C07281=1141.600,42.960,-51.075,-179.900,6.400,149.135
C07282=1141.605,42.711,-51.060,-179.904,6.398,149.135
C07283=1141.610,42.462,-51.044,-179.906,6.397,149.136
C07284=1141.615,42.212,-51.029,-179.909,6.396,149.136
C07285=1141.621,41.962,-51.014,-179.911,6.395,149.137
C07286=1141.625,41.713,-50.999,-179.914,6.394,149.138
C07287=1141.630,41.463,-50.983,-179.916,6.393,149.138
C07288=1141.635,41.214,-50.969,-179.919,6.392,149.139
C07289=1141.641,40.964,-50.953,-179.922,6.391,149.139
C07290=1141.645,40.715,-50.938,-179.924,6.390,149.140
C07291=1141.651,40.466,-50.923,-179.927,6.389,149.140
C07292=1141.656,40.216,-50.908,-179.929,6.388,149.141
C07293=1141.660,39.967,-50.893,-179.932,6.387,149.141
C07294=1141.666,39.717,-50.878,-179.935,6.386,149.142
C07295=1141.671,39.468,-50.864,-179.937,6.384,149.142
C07296=1141.676,39.218,-50.848,-179.940,6.384,149.143
C07297=1141.680,38.969,-50.833,-179.943,6.382,149.143
C07298=1141.686,38.718,-50.818,-179.945,6.381,149.144
C07299=1141.690,38.469,-50.803,-179.948,6.380,149.144
C07300=1141.696,38.219,-50.788,-179.950,6.379,149.145
C07301=1141.701,37.970,-50.773,-179.953,6.379,149.146
C07302=1141.705,37.721,-50.758,-179.956,6.377,149.146
C07303=1141.711,37.471,-50.743,-179.958,6.376,149.146
C07304=1141.716,37.222,-50.728,-179.961,6.375,149.147
C07305=1141.721,36.972,-50.713,-179.963,6.374,149.148
C07306=1141.726,36.723,-50.698,-179.966,6.372,149.148
C07307=1141.731,36.473,-50.684,-179.969,6.372,149.149
C07308=1141.736,36.224,-50.668,-179.971,6.370,149.149
C07309=1141.741,35.974,-50.654,-179.974,6.370,149.150
C07310=1141.746,35.725,-50.639,-179.976,6.369,149.150
C07311=1141.752,35.475,-50.624,-179.979,6.367,149.151
C07312=1141.756,35.226,-50.609,-179.982,6.367,149.151
C07313=1141.761,34.976,-50.595,-179.984,6.365,149.152
C07314=1141.767,34.727,-50.579,-179.987,6.365,149.152
C07315=1141.772,34.477,-50.565,-179.989,6.364,149.153
C07316=1141.776,34.228,-50.550,-179.992,6.362,149.153
C07317=1141.782,33.978,-50.535,-179.994,6.362,149.154
C07318=1141.787,33.729,-50.520,-179.997,6.360,149.155
C07319=1141.792,33.479,-50.506,-180.000,6.360,149.155
C07320=1141.797,33.230,-50.490,179.997,6.358,149.156
C07321=1141.802,32.980,-50.476,179.995,6.357,149.156
C07322=1141.807,32.730,-50.462,179.993,6.357,149.157
C07323=1141.812,32.481,-50.447,179.990,6.355,149.157
C07324=1141.817,32.231,-50.432,179.987,6.355,149.158
C07325=1141.822,31.983,-50.417,179.985,6.353,149.158
C07326=1141.827,31.733,-50.403,179.982,6.352,149.159
C07327=1141.832,31.483,-50.389,179.980,6.352,149.159
C07328=1141.838,31.234,-50.373,179.977,6.350,149.160
C07329=1141.843,30.984,-50.359,179.974,6.350,149.160
C07330=1141.848,30.735,-50.345,179.972,6.348,149.161
C07331=1141.852,30.486,-50.330,179.969,6.348,149.162
C07332=1141.858,30.236,-50.315,179.967,6.347,149.162
C07333=1141.863,29.986,-50.300,179.964,6.345,149.162
C07334=1141.868,29.737,-50.285,179.961,6.345,149.163
C07335=1141.873,29.487,-50.271,179.959,6.343,149.164
C07336=1141.878,29.237,-50.257,179.956,6.343,149.164
C07337=1141.884,28.988,-50.242,179.954,6.342,149.165
C07338=1141.888,28.739,-50.227,179.951,6.340,149.165
C07339=1141.893,28.489,-50.213,179.948,6.340,149.166
C07340=1141.898,28.239,-50.199,179.946,6.339,149.166
C07341=1141.903,27.990,-50.185,179.943,6.338,149.167
C07342=1141.908,27.721,-50.169,179.941,6.337,149.167
C07343=1141.914,27.452,-50.152,179.938,6.335,149.168
C07344=1141.920,27.182,-50.138,179.935,6.334,149.169
C07345=1141.925,26.914,-50.122,179.932,6.333,149.169
C07346=1141.930,26.665,-50.108,179.930,6.333,149.170
C07347=1141.935,26.415,-50.094,179.927,6.331,149.170
C07348=1141.940,26.166,-50.079,179.925,6.331,149.171
C07349=1141.946,25.916,-50.064,179.922,6.329,149.171
C07350=1141.951,25.666,-50.049,179.919,6.328,149.172
C07351=1141.956,25.416,-50.035,179.917,6.328,149.172
C07352=1141.961,25.167,-50.021,179.914,6.326,149.173
C07353=1141.966,24.918,-50.007,179.912,6.326,149.174
C07354=1141.971,24.668,-49.993,179.910,6.325,149.174
C07355=1141.976,24.418,-49.978,179.906,6.323,149.175
C07356=1141.981,24.169,-49.964,179.904,6.323,149.175
C07357=1141.986,23.920,-49.950,179.902,6.322,149.176
C07358=1141.991,23.670,-49.935,179.899,6.321,149.176
C07359=1141.996,23.421,-49.921,179.897,6.320,149.177
C07360=1142.001,23.171,-49.907,179.894,6.319,149.177
C07361=1142.006,22.921,-49.892,179.891,6.318,149.178
C07362=1142.012,22.672,-49.879,179.889,6.317,149.178
C07363=1142.017,22.423,-49.864,179.886,6.316,149.179
C07364=1142.022,22.173,-49.850,179.884,6.315,149.180
C07365=1142.027,21.923,-49.836,179.881,6.314,149.180
C07366=1142.032,21.674,-49.822,179.879,6.314,149.181
C07367=1142.037,21.424,-49.808,179.876,6.312,149.181
C07368=1142.042,21.175,-49.793,179.873,6.311,149.182
C07369=1142.047,20.925,-49.779,179.871,6.311,149.182
C07370=1142.052,20.675,-49.765,179.868,6.309,149.183
C07371=1142.057,20.426,-49.751,179.866,6.309,149.183
C07372=1142.062,20.177,-49.736,179.864,6.308,149.184
C07373=1142.067,19.927,-49.722,179.860,6.307,149.185
C07374=1142.073,19.677,-49.709,179.858,6.306,149.185
C07375=1142.078,19.428,-49.695,179.856,6.305,149.185
C07376=1142.083,19.178,-49.680,179.853,6.304,149.186
C07377=1142.088,18.928,-49.666,179.851,6.303,149.187
C07378=1142.094,18.679,-49.652,179.848,6.302,149.187
C07379=1142.099,18.429,-49.638,179.845,6.301,149.188
C07380=1142.103,18.180,-49.624,179.843,6.300,149.188
C07381=1142.108,17.931,-49.610,179.840,6.299,149.189
C07382=1142.113,17.681,-49.596,179.837,6.298,149.189
C07383=1142.119,17.431,-49.583,179.835,6.297,149.190
C07384=1142.124,17.181,-49.568,179.833,6.297,149.190
C07385=1142.129,16.932,-49.554,179.831,6.296,149.191
C07386=1142.134,16.683,-49.540,179.827,6.295,149.192
C07387=1142.139,16.433,-49.526,179.825,6.294,149.192
C07388=1142.144,16.184,-49.513,179.822,6.293,149.193
C07389=1142.149,15.934,-49.499,179.820,6.292,149.193
C07390=1142.154,15.684,-49.485,179.817,6.291,149.194
C07391=1142.160,15.435,-49.471,179.815,6.290,149.194
C07392=1142.165,15.185,-49.456,179.813,6.290,149.195
C07393=1142.170,14.935,-49.443,179.809,6.288,149.195
C07394=1142.175,14.686,-49.430,179.807,6.288,149.196
C07395=1142.180,14.437,-49.415,179.805,6.287,149.196
C07396=1142.185,14.188,-49.401,179.802,6.286,149.197
C07397=1142.190,13.937,-49.388,179.800,6.285,149.198
C07398=1142.195,13.688,-49.374,179.797,6.284,149.198
C07399=1142.200,13.439,-49.360,179.795,6.283,149.199
C07400=1142.205,13.189,-49.347,179.792,6.282,149.199
C07401=1142.210,12.939,-49.332,179.789,6.281,149.200
C07402=1142.216,12.690,-49.319,179.787,6.281,149.200
C07403=1142.220,12.440,-49.306,179.784,6.279,149.201
C07404=1142.226,12.191,-49.292,179.782,6.279,149.201
C07405=1142.231,11.941,-49.277,179.780,6.278,149.202
C07406=1142.236,11.691,-49.264,179.777,6.277,149.203
C07407=1142.241,11.442,-49.250,179.774,6.276,149.203
C07408=1142.246,11.192,-49.236,179.772,6.275,149.204
C07409=1142.252,10.943,-49.223,179.769,6.274,149.204
C07410=1142.256,10.693,-49.209,179.767,6.274,149.205
C07411=1142.261,10.443,-49.196,179.764,6.272,149.205
C07412=1142.267,10.194,-49.182,179.762,6.272,149.206
C07413=1142.272,9.944,-49.168,179.759,6.271,149.206
C07414=1142.277,9.695,-49.155,179.757,6.270,149.207
C07415=1142.282,9.445,-49.141,179.754,6.269,149.207
C07416=1142.288,9.196,-49.127,179.752,6.268,149.208
C07417=1142.292,8.946,-49.114,179.749,6.267,149.209
C07418=1142.298,8.697,-49.101,179.747,6.267,149.209
C07419=1142.303,8.447,-49.086,179.744,6.265,149.210
C07420=1142.307,8.197,-49.073,179.742,6.265,149.210
C07421=1142.313,7.948,-49.059,179.739,6.264,149.211
C07422=1142.318,7.698,-49.046,179.737,6.263,149.211
C07423=1142.323,7.449,-49.033,179.734,6.262,149.212
C07424=1142.328,7.198,-49.019,179.732,6.261,149.212
C07425=1142.333,6.950,-49.006,179.729,6.260,149.213
C07426=1142.338,6.699,-48.992,179.727,6.260,149.214
C07427=1142.344,6.450,-48.978,179.724,6.258,149.214
C07428=1142.348,6.200,-48.965,179.721,6.258,149.215
C07429=1142.354,5.951,-48.951,179.719,6.257,149.215
C07430=1142.358,5.701,-48.938,179.717,6.256,149.216
C07431=1142.364,5.452,-48.925,179.714,6.255,149.216
C07432=1142.369,5.202,-48.911,179.711,6.254,149.217
C07433=1142.374,4.953,-48.898,179.709,6.254,149.218
C07434=1142.379,4.703,-48.884,179.707,6.253,149.218
C07435=1142.384,4.454,-48.871,179.704,6.252,149.218
C07436=1142.390,4.203,-48.858,179.701,6.251,149.219
C07437=1142.395,3.955,-48.845,179.699,6.250,149.220
C07438=1142.400,3.704,-48.831,179.696,6.250,149.220
C07439=1142.405,3.455,-48.818,179.694,6.249,149.221
C07440=1142.410,3.205,-48.804,179.692,6.249,149.221
C07441=1142.415,2.956,-48.792,179.689,6.247,149.222
C07442=1142.421,2.706,-48.778,179.687,6.246,149.222
C07443=1142.425,2.457,-48.765,179.684,6.246,149.223
C07444=1142.431,2.207,-48.751,179.682,6.245,149.224
C07445=1142.435,1.957,-48.738,179.679,6.244,149.224
C07446=1142.442,1.689,-48.724,179.676,6.243,149.225
C07447=1142.447,1.419,-48.710,179.674,6.242,149.225
C07448=1142.453,1.149,-48.695,179.671,6.241,149.226
C07449=1142.458,0.879,-48.681,179.668,6.240,149.227
C07450=1142.464,0.630,-48.668,179.666,6.240,149.227
C07451=1142.468,0.381,-48.654,179.663,6.239,149.228
C07452=1142.474,0.131,-48.641,179.661,6.238,149.228
C07453=1142.479,-0.119,-48.628,179.658,6.237,149.229
C07454=1142.483,-0.369,-48.615,179.656,6.236,149.229
C07455=1142.489,-0.618,-48.602,179.654,6.235,149.230
C07456=1142.494,-0.867,-48.589,179.651,6.235,149.230
C07457=1142.499,-1.117,-48.575,179.648,6.233,149.231
C07458=1142.504,-1.367,-48.563,179.646,6.233,149.232
C07459=1142.510,-1.617,-48.549,179.643,6.232,149.232
C07460=1142.515,-1.866,-48.536,179.641,6.231,149.233
C07461=1142.520,-2.115,-48.523,179.639,6.231,149.233
C07462=1142.525,-2.365,-48.510,179.636,6.230,149.234
C07463=1142.530,-2.615,-48.497,179.633,6.229,149.234
C07464=1142.536,-2.864,-48.484,179.631,6.228,149.235
C07465=1142.540,-3.114,-48.471,179.629,6.227,149.235
C07466=1142.545,-3.363,-48.458,179.626,6.227,149.236
C07467=1142.551,-3.613,-48.445,179.624,6.226,149.236
C07468=1142.556,-3.863,-48.432,179.621,6.226,149.237
C07469=1142.561,-4.112,-48.419,179.619,6.224,149.238
C07470=1142.567,-4.361,-48.406,179.616,6.223,149.238
C07471=1142.571,-4.611,-48.393,179.614,6.223,149.239
C07472=1142.576,-4.861,-48.380,179.611,6.222,149.239
C07473=1142.582,-5.110,-48.367,179.609,6.222,149.240
C07474=1142.587,-5.360,-48.354,179.607,6.221,149.240
C07475=1142.592,-5.610,-48.341,179.604,6.219,149.241
C07476=1142.598,-5.859,-48.328,179.601,6.219,149.242
C07477=1142.602,-6.109,-48.315,179.599,6.218,149.242
C07478=1142.607,-6.359,-48.302,179.596,6.218,149.243
C07479=1142.613,-6.608,-48.289,179.594,6.217,149.243
C07480=1142.618,-6.858,-48.276,179.592,6.216,149.244
C07481=1142.623,-7.108,-48.264,179.589,6.216,149.244
C07482=1142.628,-7.357,-48.251,179.587,6.214,149.245
C07483=1142.634,-7.607,-48.238,179.584,6.214,149.245
C07484=1142.638,-7.857,-48.225,179.582,6.213,149.246
C07485=1142.643,-8.106,-48.212,179.580,6.212,149.246
C07486=1142.648,-8.355,-48.200,179.577,6.211,149.247
C07487=1142.654,-8.605,-48.186,179.575,6.211,149.248
C07488=1142.659,-8.855,-48.174,179.572,6.210,149.248
C07489=1142.664,-9.105,-48.162,179.569,6.209,149.249
C07490=1142.669,-9.354,-48.149,179.567,6.208,149.249
C07491=1142.675,-9.605,-48.135,179.564,6.207,149.250
C07492=1142.680,-9.854,-48.123,179.562,6.207,149.250
C07493=1142.685,-10.103,-48.110,179.560,6.206,149.251
C07494=1142.690,-10.352,-48.098,179.557,6.205,149.252
C07495=1142.695,-10.602,-48.085,179.555,6.205,149.252
C07496=1142.700,-10.852,-48.072,179.553,6.204,149.253
C07497=1142.706,-11.101,-48.059,179.550,6.203,149.253
C07498=1142.711,-11.351,-48.047,179.547,6.202,149.254
C07499=1142.716,-11.601,-48.034,179.545,6.201,149.254
C07500=1142.721,-11.851,-48.021,179.542,6.201,149.255
C07501=1142.726,-12.100,-48.009,179.540,6.200,149.255
C07502=1142.731,-12.349,-47.996,179.538,6.199,149.256
C07503=1142.737,-12.600,-47.984,179.535,6.199,149.257
C07504=1142.742,-12.849,-47.971,179.533,6.198,149.257
C07505=1142.747,-13.099,-47.958,179.530,6.198,149.258
C07506=1142.752,-13.348,-47.946,179.528,6.196,149.258
C07507=1142.757,-13.598,-47.933,179.526,6.195,149.259
C07508=1142.762,-13.847,-47.921,179.523,6.195,149.259
C07509=1142.767,-14.097,-47.909,179.521,6.194,149.260
C07510=1142.772,-14.347,-47.896,179.518,6.194,149.261
C07511=1142.778,-14.596,-47.882,179.516,6.193,149.261
C07512=1142.783,-14.846,-47.870,179.514,6.192,149.262
C07513=1142.788,-15.096,-47.858,179.511,6.192,149.262
C07514=1142.794,-15.345,-47.845,179.509,6.191,149.263
C07515=1142.799,-15.595,-47.833,179.506,6.190,149.263
C07516=1142.803,-15.845,-47.820,179.504,6.190,149.264
C07517=1142.809,-16.094,-47.808,179.501,6.188,149.264
C07518=1142.814,-16.344,-47.796,179.499,6.188,149.265
C07519=1142.819,-16.594,-47.783,179.496,6.187,149.265
C07520=1142.824,-16.843,-47.771,179.494,6.186,149.266
C07521=1142.830,-17.093,-47.759,179.492,6.186,149.267
C07522=1142.835,-17.342,-47.746,179.489,6.185,149.267
C07523=1142.840,-17.591,-47.734,179.487,6.184,149.268
C07524=1142.845,-17.842,-47.721,179.485,6.184,149.268
C07525=1142.850,-18.091,-47.709,179.482,6.183,149.269
C07526=1142.855,-18.341,-47.696,179.480,6.182,149.269
C07527=1142.860,-18.591,-47.684,179.477,6.182,149.270
C07528=1142.866,-18.840,-47.672,179.475,6.181,149.271
C07529=1142.871,-19.090,-47.660,179.472,6.180,149.271
C07530=1142.876,-19.339,-47.647,179.469,6.179,149.272
C07531=1142.881,-19.589,-47.635,179.467,6.178,149.272
C07532=1142.887,-19.838,-47.623,179.465,6.178,149.273
C07533=1142.892,-20.088,-47.610,179.462,6.177,149.273
C07534=1142.897,-20.338,-47.598,179.460,6.176,149.274
C07535=1142.902,-20.588,-47.585,179.458,6.176,149.275
C07536=1142.907,-20.838,-47.573,179.455,6.175,149.275
C07537=1142.912,-21.087,-47.561,179.453,6.174,149.276
C07538=1142.918,-21.337,-47.549,179.450,6.174,149.276
C07539=1142.923,-21.586,-47.536,179.448,6.173,149.277
C07540=1142.928,-21.836,-47.524,179.446,6.173,149.277
C07541=1142.933,-22.086,-47.512,179.443,6.172,149.278
C07542=1142.939,-22.335,-47.500,179.441,6.171,149.278
C07543=1142.944,-22.585,-47.487,179.439,6.171,149.279
C07544=1142.949,-22.835,-47.475,179.436,6.170,149.280
C07545=1142.955,-23.084,-47.463,179.434,6.170,149.280
C07546=1142.959,-23.334,-47.452,179.432,6.169,149.281
C07547=1142.965,-23.584,-47.440,179.429,6.167,149.281
C07548=1142.970,-23.833,-47.427,179.426,6.167,149.282
C07549=1142.975,-24.083,-47.415,179.424,6.166,149.282
C07550=1142.980,-24.353,-47.402,179.421,6.166,149.283
C07551=1142.987,-24.623,-47.388,179.419,6.165,149.283
C07552=1142.992,-24.893,-47.375,179.416,6.164,149.284
C07553=1142.997,-25.163,-47.362,179.414,6.164,149.285
C07554=1143.003,-25.413,-47.350,179.412,6.163,149.285
C07555=1143.008,-25.662,-47.338,179.409,6.162,149.286
C07556=1143.013,-25.912,-47.327,179.407,6.162,149.287
C07557=1143.018,-26.161,-47.314,179.404,6.160,149.287
C07558=1143.023,-26.411,-47.302,179.402,6.160,149.287
C07559=1143.029,-26.661,-47.290,179.399,6.159,149.288
C07560=1143.034,-26.911,-47.278,179.397,6.158,149.289
C07561=1143.039,-27.160,-47.266,179.394,6.158,149.289
C07562=1143.044,-27.410,-47.254,179.392,6.157,149.290
C07563=1143.049,-27.659,-47.242,179.390,6.156,149.290
C07564=1143.054,-27.909,-47.230,179.387,6.156,149.291
C07565=1143.061,-28.159,-47.218,179.385,6.155,149.291
C07566=1143.065,-28.408,-47.207,179.382,6.155,149.292
C07567=1143.070,-28.658,-47.195,179.380,6.154,149.293
C07568=1143.076,-28.908,-47.183,179.378,6.153,149.293
C07569=1143.081,-29.157,-47.171,179.375,6.153,149.294
C07570=1143.086,-29.407,-47.160,179.373,6.152,149.294
C07571=1143.091,-29.656,-47.147,179.371,6.151,149.295
C07572=1143.096,-29.906,-47.135,179.368,6.151,149.295
C07573=1143.102,-30.156,-47.123,179.366,6.150,149.296
C07574=1143.107,-30.406,-47.112,179.363,6.150,149.297
C07575=1143.112,-30.655,-47.099,179.361,6.149,149.297
C07576=1143.117,-30.905,-47.087,179.359,6.148,149.298
C07577=1143.123,-31.155,-47.075,179.356,6.148,149.298
C07578=1143.127,-31.405,-47.064,179.354,6.147,149.299
C07579=1143.133,-31.655,-47.052,179.352,6.146,149.299
C07580=1143.138,-31.903,-47.040,179.349,6.146,149.300
C07581=1143.143,-32.153,-47.029,179.347,6.145,149.300
C07582=1143.149,-32.403,-47.017,179.345,6.144,149.301
C07583=1143.154,-32.653,-47.005,179.342,6.144,149.302
C07584=1143.159,-32.902,-46.994,179.340,6.143,149.302
C07585=1143.164,-33.152,-46.982,179.338,6.142,149.303
C07586=1143.170,-33.402,-46.970,179.335,6.142,149.303
C07587=1143.174,-33.651,-46.958,179.333,6.141,149.304
C07588=1143.180,-33.901,-46.946,179.331,6.140,149.304
C07589=1143.185,-34.150,-46.935,179.328,6.140,149.305
C07590=1143.190,-34.400,-46.923,179.326,6.139,149.306
C07591=1143.195,-34.650,-46.911,179.323,6.138,149.306
C07592=1143.201,-34.900,-46.899,179.322,6.138,149.306
C07593=1143.206,-35.150,-46.888,179.319,6.138,149.307
C07594=1143.211,-35.400,-46.876,179.317,6.137,149.308
C07595=1143.217,-35.649,-46.865,179.314,6.137,149.308
C07596=1143.222,-35.898,-46.853,179.312,6.136,149.309
C07597=1143.227,-36.148,-46.842,179.310,6.135,149.309
C07598=1143.232,-36.398,-46.830,179.307,6.135,149.310
C07599=1143.237,-36.648,-46.818,179.305,6.134,149.310
C07600=1143.243,-36.898,-46.807,179.302,6.134,149.311
C07601=1143.248,-37.147,-46.796,179.300,6.133,149.312
C07602=1143.253,-37.397,-46.784,179.298,6.132,149.312
C07603=1143.258,-37.646,-46.772,179.295,6.132,149.313
C07604=1143.264,-37.896,-46.761,179.293,6.131,149.313
C07605=1143.268,-38.146,-46.749,179.291,6.130,149.314
C07606=1143.274,-38.395,-46.738,179.288,6.130,149.314
C07607=1143.280,-38.645,-46.726,179.286,6.129,149.315
C07608=1143.284,-38.895,-46.715,179.284,6.128,149.315
C07609=1143.290,-39.145,-46.703,179.281,6.128,149.316
C07610=1143.295,-39.394,-46.691,179.279,6.127,149.317
C07611=1143.301,-39.643,-46.680,179.277,6.127,149.317
C07612=1143.305,-39.893,-46.669,179.274,6.126,149.318
C07613=1143.311,-40.143,-46.657,179.272,6.125,149.318
C07614=1143.315,-40.393,-46.645,179.269,6.125,149.319
C07615=1143.321,-40.642,-46.634,179.268,6.125,149.319
C07616=1143.326,-40.892,-46.623,179.266,6.124,149.320
C07617=1143.332,-41.142,-46.611,179.263,6.123,149.321
C07618=1143.337,-41.392,-46.600,179.261,6.123,149.321
C07619=1143.343,-41.641,-46.589,179.258,6.122,149.322
C07620=1143.347,-41.891,-46.577,179.256,6.121,149.322
C07621=1143.353,-42.141,-46.565,179.254,6.121,149.323
C07622=1143.357,-42.390,-46.554,179.251,6.120,149.323
C07623=1143.364,-42.640,-46.543,179.249,6.120,149.324
C07624=1143.368,-42.890,-46.532,179.247,6.119,149.324
C07625=1143.374,-43.140,-46.520,179.244,6.118,149.325
C07626=1143.379,-43.389,-46.509,179.242,6.118,149.326
C07627=1143.384,-43.638,-46.498,179.240,6.117,149.326
C07628=1143.389,-43.888,-46.486,179.237,6.116,149.327
C07629=1143.394,-44.138,-46.476,179.235,6.116,149.327
C07630=1143.400,-44.388,-46.464,179.233,6.116,149.328
C07631=1143.405,-44.637,-46.453,179.231,6.115,149.328
C07632=1143.410,-44.887,-46.441,179.228,6.114,149.329
C07633=1143.415,-45.137,-46.430,179.226,6.114,149.330
C07634=1143.421,-45.386,-46.419,179.224,6.113,149.330
C07635=1143.426,-45.636,-46.407,179.221,6.112,149.331
C07636=1143.431,-45.886,-46.396,179.219,6.112,149.331
C07637=1143.436,-46.135,-46.386,179.217,6.111,149.332
C07638=1143.442,-46.385,-46.374,179.214,6.111,149.332
C07639=1143.447,-46.635,-46.363,179.212,6.110,149.333
C07640=1143.453,-46.884,-46.351,179.210,6.109,149.333
C07641=1143.458,-47.134,-46.341,179.207,6.110,149.334
C07642=1143.462,-47.384,-46.329,179.205,6.109,149.335
C07643=1143.468,-47.633,-46.318,179.203,6.108,149.335
C07644=1143.473,-47.883,-46.307,179.200,6.108,149.336
C07645=1143.478,-48.133,-46.296,179.198,6.107,149.336
C07646=1143.484,-48.382,-46.284,179.196,6.106,149.337
C07647=1143.489,-48.633,-46.274,179.193,6.106,149.337
C07648=1143.494,-48.882,-46.263,179.191,6.105,149.338
C07649=1143.500,-49.132,-46.252,179.189,6.104,149.338
C07650=1143.505,-49.382,-46.241,179.186,6.104,149.339
C07651=1143.509,-49.631,-46.229,179.185,6.104,149.340
C07652=1143.516,-49.881,-46.218,179.183,6.103,149.340
C07653=1143.520,-50.131,-46.207,179.180,6.103,149.341
C07654=1143.527,-50.401,-46.195,179.178,6.102,149.341
C07655=1143.532,-50.672,-46.184,179.175,6.102,149.342
C07656=1143.537,-50.943,-46.171,179.173,6.101,149.342
C07657=1143.543,-51.213,-46.159,179.170,6.100,149.343
C07658=1143.548,-51.463,-46.149,179.168,6.100,149.344
C07659=1143.554,-51.713,-46.137,179.165,6.099,149.344
C07660=1143.559,-51.963,-46.127,179.163,6.098,149.345
C07661=1143.564,-52.212,-46.115,179.161,6.098,149.345
C07662=1143.570,-52.462,-46.105,179.158,6.097,149.346
C07663=1143.575,-52.712,-46.093,179.156,6.096,149.346
C07664=1143.580,-52.961,-46.082,179.154,6.096,149.347
C07665=1143.585,-53.211,-46.072,179.152,6.096,149.348
C07666=1143.590,-53.461,-46.061,179.150,6.095,149.348
C07667=1143.596,-53.710,-46.050,179.147,6.095,149.349
C07668=1143.601,-53.960,-46.039,179.145,6.094,149.349
C07669=1143.607,-54.210,-46.028,179.143,6.093,149.350
C07670=1143.612,-54.460,-46.018,179.140,6.093,149.350
C07671=1143.616,-54.710,-46.006,179.138,6.092,149.351
C07672=1143.622,-54.959,-45.996,179.136,6.092,149.351
C07673=1143.627,-55.209,-45.984,179.134,6.091,149.352
C07674=1143.633,-55.459,-45.974,179.131,6.091,149.353
C07675=1143.638,-55.708,-45.963,179.129,6.090,149.353
C07676=1143.643,-55.958,-45.953,179.127,6.090,149.354
C07677=1143.648,-56.207,-45.941,179.124,6.089,149.354
C07678=1143.654,-56.457,-45.931,179.123,6.089,149.355
C07679=1143.659,-56.707,-45.920,179.120,6.088,149.355
C07680=1143.664,-56.957,-45.909,179.118,6.088,149.356
C07681=1143.670,-57.207,-45.898,179.116,6.087,149.356
C07682=1143.674,-57.456,-45.887,179.113,6.086,149.357
C07683=1143.680,-57.706,-45.877,179.111,6.086,149.358
C07684=1143.685,-57.956,-45.866,179.109,6.085,149.358
C07685=1143.690,-58.205,-45.855,179.107,6.085,149.359
C07686=1143.695,-58.455,-45.845,179.104,6.085,149.359
C07687=1143.701,-58.705,-45.835,179.102,6.084,149.360
C07688=1143.706,-58.955,-45.823,179.100,6.083,149.360
C07689=1143.712,-59.204,-45.813,179.097,6.083,149.361
C07690=1143.717,-59.454,-45.801,179.095,6.082,149.361
C07691=1143.722,-59.703,-45.791,179.093,6.082,149.362
C07692=1143.727,-59.954,-45.781,179.091,6.082,149.363
C07693=1143.733,-60.203,-45.770,179.089,6.081,149.363
C07694=1143.737,-60.453,-45.759,179.086,6.080,149.364
C07695=1143.743,-60.702,-45.749,179.084,6.080,149.364
C07696=1143.748,-60.953,-45.738,179.082,6.079,149.365
C07697=1143.753,-61.202,-45.727,179.080,6.079,149.365
C07698=1143.758,-61.452,-45.717,179.077,6.079,149.366
C07699=1143.764,-61.701,-45.707,179.075,6.078,149.366
C07700=1143.769,-61.951,-45.696,179.073,6.077,149.367
C07701=1143.774,-62.200,-45.685,179.070,6.077,149.368
C07702=1143.780,-62.450,-45.675,179.069,6.077,149.368
C07703=1143.785,-62.700,-45.664,179.066,6.076,149.369
C07704=1143.790,-62.950,-45.654,179.064,6.076,149.369
C07705=1143.795,-63.199,-45.643,179.062,6.075,149.370
C07706=1143.801,-63.449,-45.633,179.059,6.074,149.370
C07707=1143.806,-63.699,-45.622,179.057,6.073,149.371
C07708=1143.811,-63.949,-45.612,179.055,6.074,149.371
C07709=1143.817,-64.198,-45.602,179.053,6.073,149.372
C07710=1143.822,-64.448,-45.590,179.051,6.072,149.372
C07711=1143.827,-64.697,-45.580,179.048,6.072,149.373
C07712=1143.832,-64.948,-45.569,179.046,6.071,149.374
C07713=1143.838,-65.197,-45.559,179.044,6.071,149.374
C07714=1143.843,-65.448,-45.549,179.042,6.071,149.375
C07715=1143.848,-65.697,-45.538,179.039,6.070,149.375
C07716=1143.854,-65.947,-45.528,179.037,6.069,149.376
C07717=1143.859,-66.196,-45.517,179.035,6.069,149.376
C07718=1143.864,-66.446,-45.507,179.033,6.069,149.377
C07719=1143.869,-66.696,-45.496,179.031,6.068,149.377
C07720=1143.875,-66.946,-45.486,179.029,6.067,149.378
C07721=1143.880,-67.195,-45.476,179.026,6.067,149.379
C07722=1143.885,-67.445,-45.465,179.024,6.066,149.379
C07723=1143.891,-67.695,-45.455,179.022,6.066,149.379
C07724=1143.897,-67.944,-45.445,179.019,6.066,149.380
C07725=1143.902,-68.195,-45.434,179.017,6.065,149.381
C07726=1143.907,-68.444,-45.424,179.015,6.064,149.381
C07727=1143.913,-68.693,-45.413,179.012,6.064,149.382
C07728=1143.917,-68.943,-45.403,179.011,6.064,149.382
C07729=1143.922,-69.193,-45.393,179.009,6.063,149.383
C07730=1143.927,-69.443,-45.382,179.006,6.062,149.383
C07731=1143.933,-69.692,-45.372,179.004,6.062,149.384
C07732=1143.939,-69.942,-45.362,179.002,6.062,149.384
C07733=1143.944,-70.192,-45.351,179.000,6.061,149.385
C07734=1143.949,-70.442,-45.341,178.997,6.061,149.386
C07735=1143.955,-70.691,-45.331,178.995,6.060,149.386
C07736=1143.959,-70.941,-45.321,178.993,6.059,149.387
C07737=1143.965,-71.191,-45.311,178.991,6.060,149.387
C07738=1143.970,-71.440,-45.301,178.989,6.059,149.388
C07739=1143.975,-71.691,-45.290,178.986,6.058,149.388
C07740=1143.981,-71.940,-45.280,178.984,6.057,149.389
C07741=1143.986,-72.190,-45.270,178.982,6.058,149.390
C07742=1143.992,-72.439,-45.261,178.980,6.057,149.390
C07743=1143.997,-72.690,-45.250,178.978,6.056,149.390
C07744=1144.002,-72.939,-45.240,178.975,6.056,149.391
C07745=1144.008,-73.189,-45.230,178.974,6.056,149.392
C07746=1144.013,-73.439,-45.219,178.971,6.055,149.392
C07747=1144.018,-73.689,-45.209,178.969,6.054,149.393
C07748=1144.023,-73.938,-45.199,178.966,6.054,149.393
C07749=1144.029,-74.187,-45.189,178.965,6.054,149.394
C07750=1144.034,-74.438,-45.178,178.963,6.053,149.394
C07751=1144.039,-74.687,-45.168,178.961,6.052,149.395
C07752=1144.045,-74.937,-45.158,178.958,6.052,149.395
C07753=1144.050,-75.187,-45.149,178.956,6.052,149.396
C07754=1144.055,-75.437,-45.139,178.954,6.051,149.396
C07755=1144.061,-75.686,-45.128,178.951,6.051,149.397
C07756=1144.066,-75.936,-45.118,178.949,6.050,149.398
C07757=1144.071,-76.186,-45.108,178.948,6.050,149.398
C07758=1144.077,-76.457,-45.097,178.945,6.050,149.399
C07759=1144.083,-76.729,-45.087,178.943,6.049,149.399
C07760=1144.089,-77.000,-45.075,178.940,6.049,149.400
C07761=1144.094,-77.271,-45.065,178.938,6.048,149.401
C07762=1144.100,-77.522,-45.055,178.936,6.047,149.401
C07763=1144.105,-77.771,-45.045,178.934,6.048,149.402
C07764=1144.110,-78.020,-45.035,178.931,6.047,149.402
C07765=1144.116,-78.270,-45.025,178.929,6.046,149.403
C07766=1144.121,-78.520,-45.015,178.927,6.045,149.403
C07767=1144.127,-78.770,-45.005,178.925,6.046,149.404
C07768=1144.131,-79.020,-44.995,178.923,6.045,149.404
C07769=1144.137,-79.269,-44.985,178.921,6.044,149.405
C07770=1144.143,-79.519,-44.975,178.918,6.043,149.405
C07771=1144.148,-79.769,-44.966,178.916,6.044,149.406
C07772=1144.153,-80.019,-44.955,178.914,6.043,149.407
C07773=1144.158,-80.268,-44.945,178.912,6.042,149.407
C07774=1144.163,-80.518,-44.935,178.910,6.042,149.407
C07775=1144.169,-80.768,-44.926,178.908,6.042,149.408
C07776=1144.175,-81.017,-44.916,178.905,6.041,149.409
C07777=1144.179,-81.267,-44.906,178.903,6.040,149.409
C07778=1144.185,-81.517,-44.896,178.902,6.040,149.410
C07779=1144.190,-81.767,-44.887,178.899,6.040,149.410
C07780=1144.195,-82.016,-44.876,178.897,6.039,149.411
C07781=1144.201,-82.266,-44.867,178.895,6.039,149.411
C07782=1144.206,-82.516,-44.857,178.893,6.039,149.412
C07783=1144.211,-82.766,-44.847,178.890,6.038,149.413
C07784=1144.217,-83.016,-44.837,178.888,6.037,149.413
C07785=1144.222,-83.265,-44.828,178.887,6.037,149.413
C07786=1144.228,-83.515,-44.817,178.884,6.037,149.414
C07787=1144.233,-83.765,-44.808,178.882,6.036,149.415
C07788=1144.238,-84.014,-44.798,178.880,6.036,149.415
C07789=1144.243,-84.264,-44.788,178.878,6.036,149.416
C07790=1144.248,-84.514,-44.779,178.876,6.035,149.416
C07791=1144.254,-84.764,-44.769,178.873,6.034,149.417
C07792=1144.259,-85.014,-44.760,178.871,6.035,149.417
C07793=1144.265,-85.263,-44.750,178.869,6.034,149.418
C07794=1144.270,-85.512,-44.740,178.867,6.033,149.418
C07795=1144.276,-85.763,-44.730,178.865,6.033,149.419
C07796=1144.280,-86.013,-44.720,178.863,6.033,149.419
C07797=1144.286,-86.263,-44.711,178.861,6.032,149.420
C07798=1144.291,-86.512,-44.701,178.859,6.032,149.420
C07799=1144.297,-86.762,-44.692,178.856,6.032,149.421
C07800=1144.302,-87.012,-44.682,178.854,6.031,149.422
C07801=1144.307,-87.261,-44.672,178.852,6.030,149.422
C07802=1144.313,-87.511,-44.663,178.850,6.030,149.423
C07803=1144.318,-87.760,-44.653,178.848,6.029,149.423
C07804=1144.323,-88.011,-44.643,178.845,6.029,149.424
C07805=1144.328,-88.260,-44.633,178.844,6.029,149.424
C07806=1144.334,-88.511,-44.624,178.842,6.028,149.425
C07807=1144.339,-88.760,-44.614,178.839,6.027,149.425
C07808=1144.345,-89.010,-44.605,178.837,6.028,149.426
C07809=1144.349,-89.259,-44.595,178.835,6.027,149.426
C07810=1144.355,-89.509,-44.586,178.833,6.026,149.427
C07811=1144.360,-89.759,-44.576,178.831,6.026,149.427
C07812=1144.366,-90.009,-44.567,178.829,6.026,149.428
C07813=1144.371,-90.259,-44.558,178.827,6.025,149.429
C07814=1144.376,-90.508,-44.548,178.825,6.025,149.429
C07815=1144.382,-90.758,-44.539,178.823,6.024,149.430
C07816=1144.387,-91.007,-44.529,178.821,6.024,149.430
C07817=1144.393,-91.257,-44.519,178.819,6.024,149.431
C07818=1144.397,-91.507,-44.510,178.816,6.023,149.431
C07819=1144.403,-91.757,-44.500,178.814,6.023,149.432
C07820=1144.408,-92.007,-44.491,178.813,6.023,149.432
C07821=1144.414,-92.257,-44.481,178.810,6.022,149.433
C07822=1144.419,-92.507,-44.472,178.808,6.022,149.433
C07823=1144.424,-92.756,-44.462,178.806,6.022,149.434
C07824=1144.430,-93.006,-44.453,178.804,6.021,149.434
C07825=1144.435,-93.256,-44.444,178.802,6.020,149.435
C07826=1144.440,-93.505,-44.434,178.800,6.020,149.435
C07827=1144.446,-93.755,-44.425,178.797,6.020,149.436
C07828=1144.451,-94.005,-44.416,178.795,6.019,149.437
C07829=1144.456,-94.255,-44.406,178.794,6.019,149.437
C07830=1144.462,-94.505,-44.397,178.791,6.018,149.438
C07831=1144.467,-94.755,-44.387,178.789,6.017,149.438
C07832=1144.472,-95.004,-44.378,178.787,6.018,149.439
C07833=1144.477,-95.254,-44.369,178.785,6.017,149.439
C07834=1144.483,-95.504,-44.359,178.783,6.016,149.440
C07835=1144.488,-95.753,-44.350,178.781,6.016,149.440
C07836=1144.493,-96.003,-44.341,178.779,6.016,149.441
C07837=1144.499,-96.253,-44.331,178.777,6.016,149.441
C07838=1144.504,-96.502,-44.322,178.775,6.015,149.442
C07839=1144.509,-96.752,-44.313,178.773,6.015,149.442
C07840=1144.515,-97.002,-44.303,178.771,6.015,149.443
C07841=1144.520,-97.252,-44.294,178.769,6.014,149.443
C07842=1144.525,-97.502,-44.285,178.766,6.014,149.444
C07843=1144.531,-97.752,-44.275,178.764,6.014,149.444
C07844=1144.536,-98.002,-44.266,178.762,6.013,149.445
C07845=1144.542,-98.251,-44.258,178.760,6.012,149.445
C07846=1144.547,-98.501,-44.247,178.758,6.012,149.446
C07847=1144.553,-98.750,-44.239,178.756,6.012,149.447
C07848=1144.558,-99.000,-44.230,178.754,6.012,149.447
C07849=1144.564,-99.250,-44.220,178.752,6.011,149.448
C07850=1144.569,-99.499,-44.211,178.750,6.010,149.448
C07851=1144.574,-99.749,-44.202,178.748,6.010,149.449
C07852=1144.580,-99.999,-44.192,178.746,6.009,149.449
C07853=1144.585,-100.249,-44.184,178.743,6.009,149.450
C07854=1144.590,-100.499,-44.175,178.742,6.009,149.450
C07855=1144.595,-100.749,-44.166,178.740,6.008,149.451
C07856=1144.601,-100.998,-44.156,178.737,6.008,149.451
C07857=1144.606,-101.248,-44.147,178.736,6.008,149.452
C07858=1144.611,-101.498,-44.138,178.734,6.007,149.452
C07859=1144.616,-101.748,-44.129,178.731,6.007,149.453
C07860=1144.622,-101.998,-44.119,178.729,6.007,149.453
C07861=1144.628,-102.247,-44.111,178.727,6.006,149.454
C07862=1144.634,-102.519,-44.101,178.725,6.006,149.454
C07863=1144.639,-102.792,-44.091,178.723,6.006,149.455
C07864=1144.645,-103.064,-44.081,178.721,6.005,149.456
C07865=1144.651,-103.336,-44.071,178.718,6.004,149.456
C07866=1144.656,-103.586,-44.062,178.716,6.004,149.457
C07867=1144.662,-103.836,-44.052,178.714,6.004,149.457
C07868=1144.667,-104.086,-44.043,178.713,6.004,149.458
C07869=1144.672,-104.335,-44.035,178.710,6.003,149.458
C07870=1144.678,-104.585,-44.026,178.708,6.002,149.459
C07871=1144.683,-104.834,-44.017,178.707,6.002,149.459
C07872=1144.689,-105.085,-44.008,178.704,6.002,149.460
C07873=1144.694,-105.334,-43.999,178.702,6.002,149.460
C07874=1144.699,-105.584,-43.990,178.700,6.001,149.461
C07875=1144.704,-105.834,-43.981,178.698,6.000,149.461
C07876=1144.709,-106.084,-43.972,178.696,6.000,149.462
C07877=1144.715,-106.333,-43.963,178.694,6.000,149.462
C07878=1144.721,-106.583,-43.954,178.693,6.000,149.463
C07879=1144.726,-106.833,-43.945,178.690,5.999,149.463
C07880=1144.731,-107.083,-43.936,178.688,5.999,149.464
C07881=1144.737,-107.333,-43.927,178.686,5.999,149.465
C07882=1144.742,-107.583,-43.918,178.684,5.998,149.465
C07883=1144.747,-107.832,-43.910,178.682,5.998,149.466
C07884=1144.753,-108.082,-43.901,178.680,5.997,149.466
C07885=1144.758,-108.332,-43.892,178.678,5.996,149.467
C07886=1144.764,-108.582,-43.883,178.676,5.997,149.467
C07887=1144.769,-108.832,-43.874,178.674,5.996,149.468
C07888=1144.774,-109.081,-43.865,178.672,5.996,149.468
C07889=1144.780,-109.331,-43.856,178.670,5.995,149.469
C07890=1144.785,-109.580,-43.847,178.668,5.995,149.469
C07891=1144.790,-109.830,-43.838,178.666,5.995,149.470
C07892=1144.795,-110.080,-43.829,178.664,5.994,149.470
C07893=1144.800,-110.330,-43.821,178.662,5.994,149.471
C07894=1144.806,-110.579,-43.812,178.660,5.993,149.471
C07895=1144.811,-110.829,-43.803,178.658,5.994,149.472
C07896=1144.817,-111.079,-43.794,178.656,5.993,149.472
C07897=1144.823,-111.330,-43.785,178.654,5.992,149.473
C07898=1144.828,-111.579,-43.777,178.652,5.992,149.473
C07899=1144.834,-111.829,-43.768,178.650,5.991,149.474
C07900=1144.839,-112.078,-43.759,178.648,5.992,149.474
C07901=1144.844,-112.328,-43.750,178.646,5.991,149.475
C07902=1144.849,-112.578,-43.741,178.644,5.991,149.475
C07903=1144.854,-112.828,-43.732,178.642,5.990,149.476
C07904=1144.860,-113.077,-43.724,178.639,5.990,149.476
C07905=1144.866,-113.328,-43.716,178.638,5.990,149.477
C07906=1144.871,-113.577,-43.707,178.636,5.989,149.477
C07907=1144.876,-113.827,-43.698,178.634,5.989,149.478
C07908=1144.882,-114.076,-43.689,178.632,5.988,149.478
C07909=1144.887,-114.326,-43.681,178.630,5.988,149.479
C07910=1144.892,-114.576,-43.672,178.628,5.988,149.479
C07911=1144.898,-114.827,-43.663,178.627,5.988,149.480
C07912=1144.903,-115.076,-43.655,178.624,5.987,149.480
C07913=1144.908,-115.326,-43.646,178.622,5.987,149.481
C07914=1144.914,-115.575,-43.637,178.620,5.987,149.482
C07915=1144.919,-115.825,-43.629,178.618,5.986,149.482
C07916=1144.925,-116.075,-43.620,178.616,5.986,149.482
C07917=1144.930,-116.325,-43.611,178.614,5.985,149.483
C07918=1144.935,-116.575,-43.603,178.612,5.985,149.483
C07919=1144.941,-116.824,-43.594,178.610,5.984,149.484
C07920=1144.946,-117.074,-43.586,178.609,5.984,149.484
C07921=1144.952,-117.324,-43.577,178.606,5.984,149.485
C07922=1144.957,-117.574,-43.568,178.604,5.983,149.485
C07923=1144.963,-117.823,-43.560,178.603,5.983,149.486
C07924=1144.968,-118.074,-43.551,178.600,5.983,149.487
C07925=1144.973,-118.324,-43.542,178.598,5.983,149.487
C07926=1144.979,-118.573,-43.534,178.596,5.982,149.488
C07927=1144.984,-118.823,-43.526,178.595,5.982,149.488
C07928=1144.989,-119.073,-43.517,178.592,5.981,149.489
C07929=1144.995,-119.322,-43.509,178.591,5.981,149.489
C07930=1145.000,-119.572,-43.500,178.589,5.980,149.490
C07931=1145.005,-119.822,-43.492,178.587,5.981,149.490
C07932=1145.011,-120.071,-43.483,178.585,5.980,149.491
C07933=1145.016,-120.321,-43.474,178.583,5.979,149.491
C07934=1145.022,-120.572,-43.466,178.581,5.979,149.491
C07935=1145.027,-120.822,-43.457,178.579,5.978,149.492
C07936=1145.033,-121.071,-43.449,178.577,5.978,149.492
C07937=1145.037,-121.321,-43.441,178.575,5.978,149.493
C07938=1145.042,-121.571,-43.432,178.573,5.978,149.494
C07939=1145.048,-121.820,-43.424,178.571,5.977,149.494
C07940=1145.054,-122.070,-43.416,178.569,5.977,149.495
C07941=1145.059,-122.320,-43.407,178.567,5.977,149.495
C07942=1145.065,-122.570,-43.399,178.565,5.977,149.496
C07943=1145.070,-122.820,-43.390,178.563,5.976,149.496
C07944=1145.075,-123.069,-43.382,178.562,5.976,149.497
C07945=1145.081,-123.319,-43.374,178.559,5.975,149.497
C07946=1145.086,-123.569,-43.365,178.558,5.975,149.498
C07947=1145.092,-123.819,-43.357,178.556,5.974,149.498
C07948=1145.097,-124.069,-43.348,178.554,5.975,149.499
C07949=1145.102,-124.318,-43.339,178.552,5.974,149.499
C07950=1145.108,-124.568,-43.332,178.550,5.974,149.500
C07951=1145.113,-124.818,-43.323,178.548,5.973,149.500
C07952=1145.118,-125.068,-43.315,178.546,5.973,149.500
C07953=1145.124,-125.317,-43.307,178.544,5.972,149.501
C07954=1145.129,-125.568,-43.298,178.543,5.972,149.501
C07955=1145.134,-125.817,-43.290,178.540,5.972,149.502
C07956=1145.140,-126.067,-43.282,178.538,5.971,149.502
C07957=1145.145,-126.317,-43.273,178.536,5.971,149.503
C07958=1145.151,-126.567,-43.266,178.534,5.971,149.504
C07959=1145.156,-126.817,-43.257,178.532,5.971,149.504
C07960=1145.161,-127.065,-43.249,178.530,5.970,149.505
C07961=1145.167,-127.316,-43.240,178.529,5.970,149.505
C07962=1145.172,-127.566,-43.232,178.526,5.969,149.506
C07963=1145.178,-127.816,-43.224,178.525,5.969,149.506
C07964=1145.184,-128.066,-43.216,178.523,5.969,149.507
C07965=1145.189,-128.315,-43.208,178.521,5.969,149.507
C07966=1144.767,-128.326,-43.250,178.518,5.971,149.509
C07967=1144.762,-128.076,-43.259,178.520,5.972,149.508
C07968=1144.756,-127.827,-43.267,178.521,5.972,149.508
C07969=1144.752,-127.577,-43.275,178.524,5.973,149.507
C07970=1144.746,-127.327,-43.283,178.525,5.973,149.507
C07971=1144.740,-127.078,-43.292,178.527,5.974,149.506
C07972=1144.735,-126.827,-43.300,178.529,5.974,149.506
C07973=1144.730,-126.578,-43.308,178.531,5.974,149.505
C07974=1144.724,-126.328,-43.316,178.533,5.974,149.505
C07975=1144.719,-126.078,-43.325,178.535,5.975,149.504
C07976=1144.713,-125.828,-43.333,178.537,5.975,149.504
C07977=1144.708,-125.578,-43.342,178.539,5.976,149.503
C07978=1144.703,-125.329,-43.349,178.540,5.976,149.503
C07979=1144.698,-125.079,-43.358,178.543,5.976,149.502
C07980=1144.692,-124.829,-43.367,178.545,5.977,149.502
C07981=1144.686,-124.579,-43.375,178.546,5.977,149.501
C07982=1144.681,-124.330,-43.383,178.549,5.978,149.501
C07983=1144.676,-124.079,-43.391,178.550,5.978,149.500
C07984=1144.671,-123.830,-43.400,178.552,5.979,149.500
C07985=1144.665,-123.580,-43.408,178.554,5.979,149.499
C07986=1144.659,-123.331,-43.416,178.556,5.979,149.499
C07987=1144.654,-123.081,-43.425,178.558,5.979,149.498
C07988=1144.649,-122.830,-43.433,178.560,5.980,149.498
C07989=1144.644,-122.581,-43.441,178.562,5.980,149.497
C07990=1144.638,-122.331,-43.450,178.564,5.981,149.497
C07991=1144.633,-122.081,-43.458,178.565,5.981,149.496
C07992=1144.627,-121.832,-43.467,178.568,5.981,149.496
C07993=1144.622,-121.582,-43.475,178.570,5.981,149.495
C07994=1144.617,-121.332,-43.484,178.572,5.982,149.495
C07995=1144.611,-121.083,-43.493,178.573,5.982,149.494
C07996=1144.605,-120.832,-43.501,178.576,5.982,149.494
C07997=1144.601,-120.582,-43.509,178.577,5.982,149.493
C07998=1144.595,-120.333,-43.518,178.579,5.983,149.493
C07999=1144.590,-120.083,-43.526,178.582,5.984,149.492
C08000=1144.585,-119.833,-43.535,178.583,5.984,149.492
C08001=1144.579,-119.584,-43.543,178.585,5.985,149.491
C08002=1144.573,-119.333,-43.551,178.587,5.985,149.491
C08003=1144.568,-119.084,-43.560,178.589,5.985,149.490
C08004=1144.563,-118.834,-43.569,178.591,5.985,149.490
C08005=1144.557,-118.584,-43.577,178.593,5.986,149.489
C08006=1144.552,-118.334,-43.586,178.595,5.986,149.489
C08007=1144.547,-118.084,-43.595,178.597,5.986,149.488
C08008=1144.542,-117.835,-43.603,178.599,5.986,149.488
C08009=1144.536,-117.585,-43.611,178.601,5.987,149.487
C08010=1144.531,-117.335,-43.620,178.603,5.987,149.487
C08011=1144.525,-117.086,-43.628,178.605,5.988,149.486
C08012=1144.520,-116.836,-43.637,178.607,5.988,149.486
C08013=1144.515,-116.586,-43.645,178.609,5.988,149.485
C08014=1144.509,-116.336,-43.654,178.611,5.989,149.485
C08015=1144.504,-116.087,-43.663,178.612,5.989,149.484
C08016=1144.498,-115.837,-43.672,178.615,5.990,149.484
C08017=1144.493,-115.586,-43.680,178.616,5.990,149.483
C08018=1144.488,-115.336,-43.689,178.619,5.990,149.483
C08019=1144.482,-115.087,-43.697,178.620,5.990,149.482
C08020=1144.477,-114.837,-43.706,178.623,5.991,149.482
C08021=1144.472,-114.588,-43.715,178.625,5.992,149.481
C08022=1144.466,-114.338,-43.723,178.626,5.992,149.481
C08023=1144.460,-114.088,-43.732,178.629,5.992,149.480
C08024=1144.455,-113.838,-43.741,178.630,5.992,149.480
C08025=1144.450,-113.588,-43.750,178.632,5.993,149.479
C08026=1144.444,-113.339,-43.758,178.634,5.993,149.479
C08027=1144.439,-113.089,-43.767,178.636,5.994,149.478
C08028=1144.434,-112.839,-43.775,178.638,5.993,149.478
C08029=1144.429,-112.589,-43.784,178.641,5.994,149.477
C08030=1144.423,-112.339,-43.793,178.643,5.995,149.477
C08031=1144.418,-112.090,-43.802,178.644,5.995,149.476
C08032=1144.412,-111.840,-43.811,178.647,5.996,149.476
C08033=1144.407,-111.590,-43.820,178.648,5.995,149.475
C08034=1144.401,-111.340,-43.829,178.650,5.996,149.475
C08035=1144.396,-111.091,-43.837,178.652,5.996,149.474
C08036=1144.390,-110.840,-43.846,178.654,5.997,149.474
C08037=1144.385,-110.591,-43.855,178.657,5.997,149.473
C08038=1144.380,-110.341,-43.863,178.658,5.997,149.472
C08039=1144.375,-110.091,-43.872,178.661,5.998,149.472
C08040=1144.369,-109.842,-43.881,178.662,5.998,149.471
C08041=1144.364,-109.592,-43.890,178.664,5.999,149.471
C08042=1144.359,-109.342,-43.899,178.667,5.999,149.470
C08043=1144.353,-109.092,-43.908,178.668,5.999,149.470
C08044=1144.348,-108.842,-43.916,178.670,6.000,149.470
C08045=1144.342,-108.592,-43.926,178.672,6.000,149.469
C08046=1144.337,-108.343,-43.934,178.675,6.001,149.468
C08047=1144.331,-108.093,-43.943,178.676,6.000,149.468
C08048=1144.326,-107.843,-43.952,178.678,6.001,149.467
C08049=1144.321,-107.593,-43.961,178.681,6.002,149.467
C08050=1144.316,-107.344,-43.970,178.682,6.002,149.466
C08051=1144.311,-107.094,-43.979,178.684,6.003,149.466
C08052=1144.305,-106.845,-43.987,178.686,6.003,149.465
C08053=1144.299,-106.594,-43.997,178.689,6.003,149.465
C08054=1144.294,-106.345,-44.006,178.691,6.004,149.464
C08055=1144.289,-106.095,-44.015,178.692,6.004,149.464
C08056=1144.284,-105.845,-44.024,178.695,6.004,149.463
C08057=1144.278,-105.595,-44.033,178.696,6.004,149.463
C08058=1144.273,-105.345,-44.041,178.698,6.005,149.462
C08059=1144.267,-105.096,-44.051,178.701,6.006,149.462
C08060=1144.262,-104.846,-44.059,178.703,6.006,149.461
C08061=1144.256,-104.596,-44.068,178.705,6.006,149.461
C08062=1144.251,-104.346,-44.077,178.706,6.006,149.460
C08063=1144.246,-104.096,-44.086,178.709,6.007,149.460
C08064=1144.241,-103.846,-44.095,178.711,6.008,149.459
C08065=1144.235,-103.596,-44.105,178.712,6.008,149.459
C08066=1144.230,-103.347,-44.114,178.715,6.008,149.458
C08067=1144.224,-103.075,-44.123,178.717,6.009,149.457
C08068=1144.218,-102.803,-44.134,178.719,6.009,149.457
C08069=1144.212,-102.531,-44.143,178.722,6.009,149.456
C08070=1144.207,-102.259,-44.153,178.724,6.010,149.456
C08071=1144.202,-102.009,-44.162,178.726,6.011,149.455
C08072=1144.196,-101.759,-44.172,178.728,6.011,149.455
C08073=1144.191,-101.509,-44.181,178.730,6.011,149.454
C08074=1144.186,-101.259,-44.189,178.732,6.011,149.454
C08075=1144.180,-101.009,-44.198,178.734,6.012,149.453
C08076=1144.174,-100.760,-44.207,178.736,6.012,149.453
C08077=1144.169,-100.511,-44.217,178.738,6.012,149.452
C08078=1144.164,-100.261,-44.226,178.740,6.013,149.452
C08079=1144.159,-100.011,-44.235,178.742,6.014,149.451
C08080=1144.153,-99.761,-44.244,178.744,6.013,149.450
C08081=1144.148,-99.511,-44.253,178.747,6.014,149.450
C08082=1144.143,-99.262,-44.263,178.748,6.014,149.449
C08083=1144.137,-99.011,-44.272,178.750,6.015,149.449
C08084=1144.132,-98.762,-44.281,178.753,6.016,149.448
C08085=1144.126,-98.512,-44.290,178.754,6.016,149.448
C08086=1144.121,-98.262,-44.300,178.757,6.016,149.447
C08087=1144.116,-98.012,-44.309,178.759,6.017,149.447
C08088=1144.111,-97.763,-44.318,178.761,6.017,149.446
C08089=1144.105,-97.512,-44.328,178.763,6.018,149.446
C08090=1144.099,-97.263,-44.337,178.764,6.018,149.445
C08091=1144.095,-97.013,-44.346,178.767,6.018,149.445
C08092=1144.089,-96.763,-44.356,178.769,6.019,149.444
C08093=1144.084,-96.513,-44.365,178.771,6.019,149.444
C08094=1144.078,-96.263,-44.373,178.773,6.019,149.443
C08095=1144.073,-96.014,-44.384,178.775,6.020,149.443
C08096=1144.068,-95.764,-44.393,178.777,6.020,149.442
C08097=1144.062,-95.514,-44.402,178.780,6.020,149.442
C08098=1144.057,-95.265,-44.412,178.782,6.021,149.441
C08099=1144.051,-95.015,-44.420,178.783,6.021,149.441
C08100=1144.046,-94.766,-44.429,178.786,6.022,149.440
C08101=1144.040,-94.516,-44.439,178.788,6.023,149.440
C08102=1144.036,-94.266,-44.449,178.790,6.022,149.439
C08103=1144.030,-94.015,-44.458,178.792,6.023,149.438
C08104=1144.025,-93.766,-44.468,178.794,6.024,149.438
C08105=1144.020,-93.516,-44.477,178.796,6.024,149.437
C08106=1144.014,-93.266,-44.486,178.798,6.024,149.437
C08107=1144.009,-93.017,-44.496,178.801,6.025,149.436
C08108=1144.003,-92.767,-44.505,178.802,6.025,149.436
C08109=1143.998,-92.517,-44.515,178.804,6.026,149.435
C08110=1143.993,-92.268,-44.524,178.807,6.026,149.435
C08111=1143.987,-92.017,-44.533,178.808,6.026,149.434
C08112=1143.982,-91.768,-44.543,178.811,6.027,149.434
C08113=1143.976,-91.518,-44.552,178.813,6.027,149.433
C08114=1143.972,-91.269,-44.562,178.815,6.027,149.433
C08115=1143.966,-91.019,-44.571,178.817,6.028,149.432
C08116=1143.961,-90.769,-44.580,178.819,6.029,149.432
C08117=1143.956,-90.520,-44.590,178.821,6.028,149.431
C08118=1143.950,-90.269,-44.599,178.823,6.029,149.430
C08119=1143.945,-90.020,-44.609,178.826,6.030,149.430
C08120=1143.939,-89.770,-44.619,178.827,6.030,149.429
C08121=1143.934,-89.521,-44.628,178.830,6.030,149.429
C08122=1143.928,-89.271,-44.638,178.832,6.031,149.428
C08123=1143.923,-89.021,-44.647,178.834,6.031,149.428
C08124=1143.918,-88.771,-44.657,178.836,6.032,149.427
C08125=1143.913,-88.521,-44.667,178.838,6.033,149.427
C08126=1143.907,-88.271,-44.676,178.840,6.032,149.426
C08127=1143.902,-88.022,-44.686,178.842,6.033,149.426
C08128=1143.897,-87.772,-44.695,178.844,6.034,149.425
C08129=1143.892,-87.523,-44.705,178.846,6.034,149.425
C08130=1143.886,-87.272,-44.714,178.849,6.034,149.424
C08131=1143.881,-87.023,-44.724,178.851,6.035,149.423
C08132=1143.875,-86.773,-44.734,178.852,6.035,149.423
C08133=1143.870,-86.524,-44.743,178.855,6.036,149.422
C08134=1143.865,-86.273,-44.753,178.857,6.036,149.422
C08135=1143.860,-86.024,-44.763,178.860,6.037,149.421
C08136=1143.854,-85.773,-44.772,178.861,6.037,149.421
C08137=1143.849,-85.524,-44.782,178.863,6.037,149.420
C08138=1143.844,-85.275,-44.792,178.866,6.038,149.420
C08139=1143.838,-85.025,-44.801,178.868,6.038,149.419
C08140=1143.833,-84.775,-44.811,178.870,6.038,149.419
C08141=1143.827,-84.525,-44.821,178.872,6.039,149.418
C08142=1143.823,-84.275,-44.831,178.874,6.039,149.418
C08143=1143.817,-84.026,-44.841,178.876,6.040,149.417
C08144=1143.812,-83.776,-44.850,178.878,6.040,149.416
C08145=1143.806,-83.526,-44.860,178.881,6.041,149.416
C08146=1143.801,-83.277,-44.870,178.882,6.041,149.416
C08147=1143.796,-83.027,-44.879,178.885,6.041,149.415
C08148=1143.791,-82.777,-44.890,178.887,6.042,149.414
C08149=1143.785,-82.527,-44.898,178.889,6.042,149.414
C08150=1143.780,-82.277,-44.909,178.891,6.043,149.413
C08151=1143.774,-82.028,-44.919,178.894,6.043,149.413
C08152=1143.769,-81.778,-44.928,178.896,6.044,149.412
C08153=1143.763,-81.528,-44.938,178.897,6.044,149.412
C08154=1143.758,-81.278,-44.949,178.900,6.045,149.411
C08155=1143.754,-81.029,-44.958,178.902,6.045,149.410
C08156=1143.748,-80.779,-44.968,178.904,6.045,149.410
C08157=1143.742,-80.529,-44.978,178.906,6.046,149.410
C08158=1143.737,-80.280,-44.987,178.908,6.047,149.409
C08159=1143.732,-80.029,-44.997,178.911,6.047,149.408
C08160=1143.726,-79.779,-45.008,178.912,6.047,149.408
C08161=1143.721,-79.530,-45.017,178.915,6.048,149.407
C08162=1143.716,-79.281,-45.027,178.917,6.049,149.407
C08163=1143.710,-79.031,-45.037,178.919,6.048,149.406
C08164=1143.706,-78.781,-45.047,178.921,6.049,149.406
C08165=1143.700,-78.531,-45.057,178.923,6.050,149.405
C08166=1143.694,-78.282,-45.067,178.926,6.050,149.405
C08167=1143.689,-78.032,-45.076,178.928,6.050,149.404
C08168=1143.684,-77.782,-45.086,178.930,6.051,149.404
C08169=1143.679,-77.532,-45.097,178.932,6.052,149.403
C08170=1143.673,-77.282,-45.107,178.934,6.052,149.403
C08171=1143.668,-77.010,-45.117,178.937,6.053,149.402
C08172=1143.662,-76.740,-45.128,178.938,6.053,149.401
C08173=1143.656,-76.468,-45.139,178.941,6.053,149.401
C08174=1143.651,-76.197,-45.150,178.943,6.054,149.400
C08175=1143.645,-75.947,-45.160,178.946,6.054,149.399
C08176=1143.639,-75.697,-45.170,178.948,6.055,149.399
C08177=1143.634,-75.448,-45.180,178.950,6.055,149.399
C08178=1143.629,-75.198,-45.190,178.952,6.056,149.398
C08179=1143.624,-74.948,-45.201,178.955,6.056,149.397
C08180=1143.618,-74.699,-45.211,178.957,6.057,149.397
C08181=1143.613,-74.449,-45.221,178.958,6.057,149.396
C08182=1143.607,-74.198,-45.231,178.961,6.058,149.396
C08183=1143.602,-73.949,-45.240,178.963,6.058,149.395
C08184=1143.597,-73.699,-45.251,178.965,6.059,149.395
C08185=1143.592,-73.449,-45.261,178.967,6.059,149.394
C08186=1143.586,-73.200,-45.271,178.970,6.059,149.393
C08187=1143.581,-72.950,-45.282,178.972,6.060,149.393
C08188=1143.576,-72.701,-45.291,178.974,6.061,149.393
C08189=1143.571,-72.451,-45.302,178.976,6.061,149.392
C08190=1143.565,-72.201,-45.312,178.978,6.061,149.391
C08191=1143.560,-71.952,-45.322,178.981,6.062,149.391
C08192=1143.555,-71.701,-45.333,178.983,6.063,149.390
C08193=1143.549,-71.452,-45.343,178.985,6.063,149.390
C08194=1143.544,-71.203,-45.353,178.987,6.063,149.389
C08195=1143.539,-70.952,-45.363,178.989,6.064,149.389
C08196=1143.534,-70.703,-45.373,178.991,6.064,149.388
C08197=1143.528,-70.453,-45.384,178.994,6.065,149.388
C08198=1143.523,-70.203,-45.394,178.996,6.065,149.387
C08199=1143.517,-69.953,-45.404,178.998,6.066,149.387
C08200=1143.512,-69.704,-45.415,179.001,6.066,149.386
C08201=1143.507,-69.454,-45.425,179.003,6.067,149.385
C08202=1143.502,-69.204,-45.435,179.005,6.067,149.385
C08203=1143.496,-68.955,-45.445,179.006,6.067,149.384
C08204=1143.491,-68.705,-45.456,179.009,6.068,149.384
C08205=1143.486,-68.455,-45.466,179.011,6.069,149.383
C08206=1143.480,-68.206,-45.476,179.014,6.069,149.383
C08207=1143.475,-67.955,-45.487,179.016,6.069,149.382
C08208=1143.469,-67.706,-45.497,179.018,6.070,149.382
C08209=1143.464,-67.456,-45.507,179.020,6.070,149.381
C08210=1143.459,-67.206,-45.518,179.022,6.071,149.381
C08211=1143.453,-66.956,-45.528,179.025,6.072,149.380
C08212=1143.449,-66.707,-45.538,179.026,6.072,149.379
C08213=1143.444,-66.458,-45.549,179.029,6.072,149.379
C08214=1143.438,-66.208,-45.559,179.031,6.073,149.378
C08215=1143.433,-65.958,-45.569,179.034,6.074,149.378
C08216=1143.428,-65.708,-45.580,179.036,6.074,149.377
C08217=1143.423,-65.458,-45.590,179.038,6.074,149.377
C08218=1143.417,-65.208,-45.600,179.040,6.075,149.376
C08219=1143.411,-64.959,-45.611,179.042,6.075,149.376
C08220=1143.407,-64.709,-45.622,179.044,6.076,149.375
C08221=1143.401,-64.460,-45.632,179.047,6.077,149.374
C08222=1143.396,-64.210,-45.643,179.049,6.077,149.374
C08223=1143.390,-63.960,-45.653,179.051,6.077,149.373
C08224=1143.385,-63.710,-45.663,179.053,6.078,149.373
C08225=1143.380,-63.460,-45.674,179.056,6.079,149.372
C08226=1143.375,-63.211,-45.685,179.058,6.079,149.372
C08227=1143.370,-62.961,-45.695,179.061,6.080,149.371
C08228=1143.364,-62.711,-45.705,179.062,6.080,149.371
C08229=1143.359,-62.461,-45.716,179.064,6.080,149.370
C08230=1143.354,-62.212,-45.727,179.067,6.081,149.369
C08231=1143.349,-61.962,-45.737,179.069,6.082,149.369
C08232=1143.343,-61.713,-45.748,179.071,6.082,149.368
C08233=1143.338,-61.462,-45.758,179.073,6.082,149.368
C08234=1143.333,-61.213,-45.769,179.076,6.083,149.367
C08235=1143.327,-60.964,-45.779,179.078,6.083,149.367
C08236=1143.322,-60.714,-45.790,179.080,6.084,149.366
C08237=1143.317,-60.464,-45.800,179.083,6.085,149.366
C08238=1143.311,-60.214,-45.812,179.085,6.085,149.365
C08239=1143.306,-59.965,-45.822,179.086,6.085,149.365
C08240=1143.301,-59.714,-45.833,179.089,6.086,149.364
C08241=1143.295,-59.465,-45.844,179.091,6.087,149.363
C08242=1143.290,-59.215,-45.854,179.093,6.087,149.363
C08243=1143.285,-58.966,-45.865,179.096,6.088,149.362
C08244=1143.280,-58.716,-45.876,179.098,6.088,149.362
C08245=1143.274,-58.466,-45.886,179.100,6.088,149.361
C08246=1143.269,-58.216,-45.897,179.103,6.089,149.361
C08247=1143.264,-57.967,-45.908,179.105,6.090,149.360
C08248=1143.259,-57.717,-45.918,179.107,6.090,149.360
C08249=1143.253,-57.467,-45.929,179.110,6.091,149.359
C08250=1143.248,-57.218,-45.940,179.112,6.092,149.358
C08251=1143.242,-56.968,-45.950,179.114,6.092,149.358
C08252=1143.238,-56.718,-45.962,179.116,6.092,149.357
C08253=1143.233,-56.468,-45.972,179.118,6.093,149.357
C08254=1143.227,-56.219,-45.982,179.120,6.094,149.356
C08255=1143.223,-55.969,-45.994,179.123,6.094,149.356
C08256=1143.216,-55.719,-46.005,179.125,6.095,149.355
C08257=1143.211,-55.469,-46.016,179.128,6.095,149.355
C08258=1143.206,-55.220,-46.026,179.130,6.095,149.354
C08259=1143.201,-54.970,-46.037,179.132,6.096,149.353
C08260=1143.196,-54.721,-46.048,179.134,6.097,149.353
C08261=1143.191,-54.471,-46.059,179.137,6.097,149.352
C08262=1143.185,-54.221,-46.070,179.139,6.098,149.352
C08263=1143.180,-53.972,-46.081,179.141,6.099,149.351
C08264=1143.175,-53.721,-46.092,179.144,6.099,149.351
C08265=1143.170,-53.472,-46.102,179.146,6.100,149.350
C08266=1143.165,-53.222,-46.113,179.147,6.100,149.350
C08267=1143.159,-52.973,-46.125,179.150,6.100,149.349
C08268=1143.154,-52.723,-46.135,179.152,6.101,149.348
C08269=1143.149,-52.473,-46.146,179.155,6.102,149.348
C08270=1143.143,-52.224,-46.157,179.157,6.102,149.347
C08271=1143.138,-51.974,-46.169,179.159,6.103,149.347
C08272=1143.132,-51.724,-46.179,179.162,6.104,149.346
C08273=1143.128,-51.474,-46.190,179.164,6.104,149.346
C08274=1143.123,-51.224,-46.201,179.166,6.104,149.345
C08275=1143.116,-50.954,-46.212,179.168,6.104,149.344
C08276=1143.111,-50.683,-46.225,179.171,6.105,149.344
C08277=1143.105,-50.412,-46.237,179.174,6.106,149.343
C08278=1143.099,-50.142,-46.249,179.176,6.107,149.343
C08279=1143.094,-49.892,-46.260,179.178,6.107,149.342
C08280=1143.089,-49.643,-46.270,179.180,6.107,149.342
C08281=1143.084,-49.393,-46.282,179.183,6.108,149.341
C08282=1143.078,-49.142,-46.293,179.185,6.109,149.340
C08283=1143.073,-48.893,-46.304,179.187,6.109,149.340
C08284=1143.068,-48.644,-46.315,179.190,6.110,149.339
C08285=1143.062,-48.393,-46.326,179.192,6.111,149.339
C08286=1143.057,-48.144,-46.337,179.194,6.111,149.338
C08287=1143.052,-47.895,-46.348,179.197,6.112,149.338
C08288=1143.047,-47.644,-46.360,179.199,6.113,149.337
C08289=1143.041,-47.395,-46.371,179.201,6.113,149.337
C08290=1143.037,-47.146,-46.382,179.203,6.113,149.336
C08291=1143.031,-46.895,-46.393,179.206,6.114,149.335
C08292=1143.026,-46.646,-46.404,179.208,6.114,149.335
C08293=1143.020,-46.396,-46.416,179.210,6.115,149.334
C08294=1143.016,-46.147,-46.427,179.213,6.116,149.334
C08295=1143.010,-45.897,-46.437,179.215,6.116,149.333
C08296=1143.005,-45.647,-46.449,179.218,6.117,149.333
C08297=1143.000,-45.397,-46.460,179.220,6.118,149.332
C08298=1142.994,-45.148,-46.471,179.222,6.118,149.332
C08299=1142.989,-44.898,-46.483,179.225,6.119,149.331
C08300=1142.984,-44.648,-46.494,179.226,6.119,149.330
C08301=1142.978,-44.399,-46.505,179.229,6.120,149.330
C08302=1142.973,-44.149,-46.517,179.231,6.120,149.329
C08303=1142.968,-43.899,-46.528,179.233,6.121,149.329
C08304=1142.963,-43.649,-46.539,179.236,6.122,149.328
C08305=1142.958,-43.400,-46.550,179.238,6.122,149.328
C08306=1142.952,-43.150,-46.562,179.240,6.123,149.327
C08307=1142.948,-42.901,-46.573,179.243,6.123,149.327
C08308=1142.941,-42.651,-46.584,179.245,6.124,149.326
C08309=1142.937,-42.401,-46.595,179.247,6.125,149.326
C08310=1142.931,-42.151,-46.607,179.250,6.125,149.325
C08311=1142.926,-41.902,-46.618,179.252,6.126,149.324
C08312=1142.920,-41.653,-46.630,179.254,6.127,149.324
C08313=1142.916,-41.403,-46.641,179.257,6.126,149.323
C08314=1142.910,-41.152,-46.652,179.259,6.127,149.323
C08315=1142.905,-40.903,-46.664,179.261,6.128,149.322
C08316=1142.899,-40.653,-46.675,179.264,6.128,149.321
C08317=1142.895,-40.404,-46.687,179.266,6.129,149.321
C08318=1142.889,-40.154,-46.698,179.268,6.130,149.321
C08319=1142.884,-39.904,-46.710,179.271,6.130,149.320
C08320=1142.879,-39.654,-46.722,179.273,6.131,149.319
C08321=1142.874,-39.405,-46.733,179.275,6.131,149.319
C08322=1142.868,-39.156,-46.744,179.278,6.132,149.318
C08323=1142.864,-38.906,-46.756,179.280,6.133,149.318
C08324=1142.858,-38.656,-46.768,179.283,6.133,149.317
C08325=1142.853,-38.407,-46.779,179.285,6.134,149.317
C08326=1142.847,-38.156,-46.790,179.287,6.135,149.316
C08327=1142.842,-37.907,-46.801,179.290,6.135,149.315
C08328=1142.837,-37.657,-46.813,179.292,6.136,149.315
C08329=1142.832,-37.407,-46.825,179.294,6.136,149.314
C08330=1142.826,-37.158,-46.836,179.297,6.137,149.314
C08331=1142.821,-36.908,-46.848,179.299,6.138,149.313
C08332=1142.816,-36.658,-46.859,179.301,6.138,149.313
C08333=1142.811,-36.409,-46.871,179.304,6.139,149.312
C08334=1142.805,-36.159,-46.883,179.305,6.139,149.312
C08335=1142.801,-35.910,-46.895,179.308,6.140,149.311
C08336=1142.795,-35.660,-46.906,179.310,6.140,149.310
C08337=1142.790,-35.411,-46.917,179.312,6.141,149.310
C08338=1142.785,-35.161,-46.929,179.315,6.142,149.309
C08339=1142.779,-34.911,-46.941,179.317,6.142,149.309
C08340=1142.775,-34.661,-46.953,179.320,6.143,149.308
C08341=1142.769,-34.411,-46.964,179.322,6.144,149.308
C08342=1142.763,-34.162,-46.976,179.324,6.144,149.307
C08343=1142.759,-33.912,-46.987,179.327,6.145,149.306
C08344=1142.753,-33.662,-46.999,179.329,6.146,149.306
C08345=1142.748,-33.413,-47.010,179.332,6.146,149.305
C08346=1142.743,-33.163,-47.022,179.334,6.147,149.305
C08347=1142.738,-32.914,-47.035,179.336,6.148,149.304
C08348=1142.732,-32.664,-47.047,179.339,6.148,149.304
C08349=1142.728,-32.414,-47.058,179.341,6.149,149.303
C08350=1142.722,-32.164,-47.070,179.343,6.150,149.303
C08351=1142.716,-31.915,-47.081,179.346,6.150,149.302
C08352=1142.712,-31.665,-47.093,179.348,6.151,149.301
C08353=1142.706,-31.415,-47.105,179.351,6.151,149.301
C08354=1142.701,-31.166,-47.117,179.353,6.152,149.300
C08355=1142.696,-30.916,-47.129,179.355,6.153,149.300
C08356=1142.691,-30.666,-47.140,179.358,6.153,149.299
C08357=1142.685,-30.417,-47.152,179.360,6.154,149.299
C08358=1142.680,-30.167,-47.164,179.362,6.155,149.298
C08359=1142.676,-29.918,-47.176,179.365,6.155,149.297
C08360=1142.670,-29.668,-47.188,179.367,6.156,149.297
C08361=1142.665,-29.418,-47.200,179.369,6.156,149.296
C08362=1142.659,-29.168,-47.212,179.372,6.157,149.296
C08363=1142.654,-28.919,-47.223,179.374,6.158,149.295
C08364=1142.649,-28.670,-47.235,179.377,6.158,149.295
C08365=1142.644,-28.420,-47.247,179.379,6.159,149.294
C08366=1142.638,-28.170,-47.259,179.381,6.159,149.293
C08367=1142.634,-27.921,-47.271,179.384,6.160,149.293
C08368=1142.628,-27.671,-47.283,179.386,6.161,149.293
C08369=1142.623,-27.421,-47.295,179.388,6.161,149.292
C08370=1142.618,-27.171,-47.307,179.391,6.162,149.291
C08371=1142.612,-26.922,-47.319,179.393,6.163,149.291
C08372=1142.608,-26.672,-47.331,179.395,6.163,149.290
C08373=1142.602,-26.423,-47.343,179.398,6.164,149.290
C08374=1142.597,-26.173,-47.355,179.400,6.165,149.289
C08375=1142.592,-25.923,-47.367,179.402,6.165,149.289
C08376=1142.586,-25.673,-47.380,179.405,6.166,149.288
C08377=1142.582,-25.424,-47.391,179.407,6.167,149.287
C08378=1142.576,-25.174,-47.403,179.410,6.168,149.287
C08379=1142.571,-24.904,-47.416,179.413,6.169,149.286
C08380=1142.565,-24.634,-47.430,179.415,6.169,149.286
C08381=1142.559,-24.364,-47.443,179.418,6.170,149.285
C08382=1142.554,-24.093,-47.456,179.420,6.171,149.285
C08383=1142.549,-23.844,-47.468,179.422,6.171,149.284
C08384=1142.544,-23.594,-47.480,179.425,6.172,149.283
C08385=1142.538,-23.344,-47.492,179.427,6.172,149.283
C08386=1142.533,-23.095,-47.505,179.430,6.174,149.282
C08387=1142.528,-22.845,-47.516,179.432,6.175,149.282
C08388=1142.523,-22.596,-47.528,179.435,6.175,149.281
C08389=1142.518,-22.346,-47.540,179.437,6.176,149.281
C08390=1142.513,-22.097,-47.553,179.440,6.176,149.280
C08391=1142.507,-21.847,-47.565,179.442,6.177,149.279
C08392=1142.502,-21.597,-47.577,179.444,6.178,149.279
C08393=1142.497,-21.348,-47.589,179.447,6.178,149.278
C08394=1142.492,-21.098,-47.602,179.449,6.179,149.278
C08395=1142.486,-20.848,-47.614,179.452,6.179,149.277
C08396=1142.481,-20.599,-47.626,179.454,6.180,149.277
C08397=1142.476,-20.349,-47.638,179.456,6.181,149.276
C08398=1142.470,-20.100,-47.651,179.459,6.181,149.275
C08399=1142.465,-19.850,-47.663,179.461,6.182,149.275
C08400=1142.460,-19.600,-47.675,179.463,6.183,149.274
C08401=1142.455,-19.350,-47.688,179.466,6.184,149.274
C08402=1142.450,-19.100,-47.700,179.468,6.184,149.273
C08403=1142.445,-18.851,-47.713,179.471,6.186,149.273
C08404=1142.439,-18.601,-47.725,179.473,6.186,149.272
C08405=1142.434,-18.352,-47.737,179.476,6.187,149.271
C08406=1142.429,-18.102,-47.749,179.478,6.188,149.271
C08407=1142.424,-17.853,-47.762,179.480,6.188,149.271
C08408=1142.419,-17.603,-47.774,179.483,6.189,149.270
C08409=1142.413,-17.353,-47.786,179.485,6.190,149.269
C08410=1142.408,-17.104,-47.799,179.487,6.190,149.269
C08411=1142.403,-16.854,-47.812,179.490,6.191,149.268
C08412=1142.398,-16.604,-47.824,179.492,6.192,149.268
C08413=1142.393,-16.355,-47.836,179.495,6.192,149.267
C08414=1142.388,-16.105,-47.849,179.497,6.193,149.267
C08415=1142.382,-15.856,-47.861,179.499,6.194,149.266
C08416=1142.377,-15.606,-47.873,179.502,6.195,149.265
C08417=1142.372,-15.357,-47.886,179.505,6.196,149.265
C08418=1142.367,-15.106,-47.898,179.507,6.196,149.264
C08419=1142.362,-14.857,-47.911,179.509,6.197,149.264
C08420=1142.356,-14.607,-47.924,179.512,6.198,149.263
C08421=1142.351,-14.358,-47.937,179.514,6.198,149.263
C08422=1142.346,-14.108,-47.949,179.516,6.199,149.262
C08423=1142.341,-13.859,-47.961,179.519,6.199,149.261
C08424=1142.336,-13.609,-47.974,179.521,6.200,149.261
C08425=1142.331,-13.359,-47.987,179.524,6.201,149.261
C08426=1142.326,-13.109,-47.999,179.527,6.202,149.260
C08427=1142.320,-12.860,-48.011,179.529,6.203,149.259
C08428=1142.315,-12.611,-48.024,179.532,6.203,149.259
C08429=1142.310,-12.361,-48.037,179.534,6.204,149.258
C08430=1142.305,-12.111,-48.049,179.536,6.205,149.258
C08431=1142.299,-11.861,-48.062,179.539,6.205,149.257
C08432=1142.294,-11.612,-48.074,179.541,6.206,149.257
C08433=1142.289,-11.363,-48.087,179.543,6.206,149.256
C08434=1142.285,-11.113,-48.100,179.546,6.208,149.255
C08435=1142.279,-10.863,-48.113,179.548,6.209,149.255
C08436=1142.274,-10.614,-48.126,179.551,6.209,149.254
C08437=1142.268,-10.364,-48.138,179.553,6.210,149.254
C08438=1142.264,-10.114,-48.151,179.556,6.211,149.253
C08439=1142.259,-9.864,-48.163,179.558,6.211,149.253
C08440=1142.254,-9.615,-48.176,179.560,6.212,149.252
C08441=1142.248,-9.365,-48.189,179.563,6.213,149.251
C08442=1142.243,-9.115,-48.202,179.566,6.214,149.251
C08443=1142.238,-8.866,-48.215,179.568,6.215,149.250
C08444=1142.233,-8.617,-48.227,179.571,6.215,149.250
C08445=1142.227,-8.367,-48.240,179.573,6.216,149.249
C08446=1142.223,-8.117,-48.253,179.575,6.217,149.249
C08447=1142.217,-7.868,-48.266,179.578,6.217,149.248
C08448=1142.212,-7.618,-48.278,179.580,6.218,149.248
C08449=1142.207,-7.368,-48.291,179.582,6.219,149.247
C08450=1142.202,-7.118,-48.304,179.585,6.220,149.247
C08451=1142.196,-6.869,-48.317,179.588,6.221,149.246
C08452=1142.191,-6.620,-48.329,179.590,6.221,149.245
C08453=1142.186,-6.369,-48.343,179.593,6.222,149.245
C08454=1142.181,-6.120,-48.355,179.595,6.223,149.244
C08455=1142.176,-5.871,-48.368,179.597,6.223,149.244
C08456=1142.171,-5.620,-48.382,179.600,6.225,149.243
C08457=1142.165,-5.371,-48.394,179.602,6.226,149.243
C08458=1142.160,-5.122,-48.407,179.605,6.226,149.242
C08459=1142.155,-4.872,-48.421,179.607,6.227,149.241
C08460=1142.150,-4.623,-48.434,179.609,6.228,149.241
C08461=1142.145,-4.373,-48.446,179.612,6.228,149.240
C08462=1142.140,-4.123,-48.460,179.615,6.230,149.240
C08463=1142.135,-3.874,-48.472,179.618,6.230,149.239
C08464=1142.130,-3.624,-48.485,179.620,6.231,149.239
C08465=1142.124,-3.374,-48.499,179.622,6.232,149.238
C08466=1142.119,-3.125,-48.511,179.625,6.232,149.238
C08467=1142.114,-2.875,-48.524,179.627,6.233,149.237
C08468=1142.109,-2.625,-48.537,179.630,6.234,149.236
C08469=1142.104,-2.376,-48.551,179.632,6.235,149.236
C08470=1142.098,-2.127,-48.564,179.634,6.236,149.235
C08471=1142.094,-1.877,-48.577,179.637,6.236,149.235
C08472=1142.089,-1.627,-48.589,179.639,6.237,149.234
C08473=1142.083,-1.378,-48.603,179.642,6.237,149.234
C08474=1142.078,-1.128,-48.616,179.645,6.239,149.233
C08475=1142.072,-0.878,-48.629,179.647,6.240,149.233
C08476=1142.068,-0.629,-48.642,179.649,6.240,149.232
C08477=1142.063,-0.379,-48.655,179.652,6.241,149.232
C08478=1142.057,-0.130,-48.668,179.654,6.241,149.231
C08479=1142.053,0.120,-48.681,179.657,6.243,149.230
C08480=1142.047,0.369,-48.695,179.659,6.244,149.230
C08481=1142.042,0.619,-48.708,179.662,6.244,149.229
C08482=1142.037,0.869,-48.721,179.664,6.245,149.229
C08483=1142.032,1.139,-48.735,179.667,6.245,149.228
C08484=1142.026,1.407,-48.750,179.670,6.247,149.228
C08485=1142.020,1.677,-48.764,179.672,6.248,149.227
C08486=1142.015,1.946,-48.778,179.675,6.249,149.226
C08487=1142.009,2.196,-48.792,179.678,6.250,149.226
C08488=1142.005,2.446,-48.804,179.680,6.250,149.225
C08489=1141.999,2.695,-48.818,179.682,6.251,149.225
C08490=1141.995,2.945,-48.831,179.685,6.252,149.224
C08491=1141.989,3.195,-48.845,179.688,6.253,149.223
C08492=1141.984,3.443,-48.858,179.690,6.254,149.223
C08493=1141.979,3.694,-48.871,179.692,6.254,149.223
C08494=1141.973,3.943,-48.885,179.695,6.255,149.222
C08495=1141.969,4.193,-48.898,179.698,6.256,149.221
C08496=1141.963,4.442,-48.911,179.700,6.257,149.221
C08497=1141.958,4.692,-48.924,179.702,6.258,149.220
C08498=1141.953,4.941,-48.938,179.705,6.259,149.220
C08499=1141.948,5.192,-48.951,179.707,6.259,149.219
C08500=1141.943,5.441,-48.965,179.710,6.261,149.219
C08501=1141.938,5.691,-48.978,179.713,6.261,149.218
C08502=1141.932,5.940,-48.991,179.715,6.262,149.217
C08503=1141.927,6.190,-49.006,179.717,6.263,149.217
C08504=1141.922,6.439,-49.018,179.720,6.264,149.216
C08505=1141.917,6.689,-49.033,179.723,6.265,149.216
C08506=1141.912,6.938,-49.045,179.725,6.265,149.215
C08507=1141.907,7.188,-49.059,179.727,6.266,149.215
C08508=1141.901,7.438,-49.073,179.730,6.268,149.214
C08509=1141.897,7.687,-49.086,179.733,6.268,149.214
C08510=1141.891,7.937,-49.100,179.735,6.269,149.213
C08511=1141.886,8.186,-49.114,179.738,6.269,149.212
C08512=1141.881,8.436,-49.126,179.740,6.270,149.212
C08513=1141.876,8.685,-49.141,179.743,6.272,149.211
C08514=1141.871,8.936,-49.154,179.745,6.272,149.211
C08515=1141.866,9.184,-49.168,179.747,6.273,149.210
C08516=1141.861,9.435,-49.181,179.750,6.273,149.210
C08517=1141.855,9.684,-49.195,179.753,6.275,149.209
C08518=1141.851,9.934,-49.208,179.755,6.276,149.209
C08519=1141.845,10.183,-49.222,179.758,6.276,149.208
C08520=1141.840,10.432,-49.236,179.760,6.278,149.208
C08521=1141.835,10.682,-49.249,179.763,6.278,149.207
C08522=1141.830,10.931,-49.263,179.765,6.279,149.206
C08523=1141.825,11.182,-49.277,179.767,6.280,149.206
C08524=1141.820,11.430,-49.290,179.771,6.281,149.205
C08525=1141.815,11.680,-49.304,179.773,6.282,149.205
C08526=1141.809,11.930,-49.317,179.775,6.282,149.204
C08527=1141.804,12.180,-49.332,179.778,6.283,149.204
C08528=1141.800,12.429,-49.345,179.780,6.285,149.203
C08529=1141.794,12.679,-49.359,179.783,6.285,149.203
C08530=1141.789,12.928,-49.373,179.785,6.286,149.202
C08531=1141.784,13.177,-49.387,179.788,6.286,149.201
C08532=1141.779,13.427,-49.400,179.791,6.288,149.201
C08533=1141.774,13.677,-49.414,179.793,6.289,149.200
C08534=1141.769,13.926,-49.428,179.795,6.289,149.200
C08535=1141.763,14.176,-49.441,179.798,6.291,149.199
C08536=1141.758,14.426,-49.456,179.801,6.291,149.199
C08537=1141.754,14.675,-49.469,179.803,6.292,149.198
C08538=1141.749,14.924,-49.483,179.805,6.293,149.198
C08539=1141.743,15.175,-49.497,179.808,6.294,149.197
C08540=1141.738,15.424,-49.511,179.811,6.295,149.197
C08541=1141.733,15.674,-49.525,179.813,6.296,149.196
C08542=1141.728,15.923,-49.539,179.816,6.297,149.195
C08543=1141.723,16.173,-49.552,179.818,6.298,149.195
C08544=1141.718,16.422,-49.566,179.821,6.298,149.194
C08545=1141.713,16.672,-49.581,179.824,6.300,149.194
C08546=1141.707,16.921,-49.594,179.826,6.300,149.193
C08547=1141.702,17.171,-49.609,179.828,6.301,149.193
C08548=1141.697,17.421,-49.622,179.831,6.302,149.192
C08549=1141.692,17.670,-49.636,179.834,6.303,149.192
C08550=1141.687,17.919,-49.650,179.836,6.304,149.191
C08551=1141.682,18.169,-49.664,179.839,6.305,149.190
C08552=1141.677,18.418,-49.678,179.842,6.306,149.190
C08553=1141.672,18.668,-49.692,179.844,6.307,149.190
C08554=1141.667,18.918,-49.707,179.846,6.307,149.189
C08555=1141.662,19.167,-49.721,179.849,6.309,149.188
C08556=1141.656,19.417,-49.734,179.851,6.310,149.188
C08557=1141.651,19.667,-49.748,179.854,6.310,149.187
C08558=1141.646,19.916,-49.763,179.857,6.312,149.187
C08559=1141.641,20.165,-49.777,179.859,6.312,149.186
C08560=1141.636,20.415,-49.791,179.862,6.313,149.186
C08561=1141.631,20.665,-49.805,179.864,6.315,149.185
C08562=1141.626,20.914,-49.819,179.867,6.315,149.185
C08563=1141.620,21.163,-49.833,179.869,6.316,149.184
C08564=1141.615,21.413,-49.848,179.872,6.317,149.183
C08565=1141.611,21.663,-49.861,179.875,6.318,149.183
C08566=1141.606,21.912,-49.876,179.877,6.319,149.182
C08567=1141.601,22.161,-49.889,179.880,6.320,149.182
C08568=1141.596,22.411,-49.904,179.882,6.321,149.181
C08569=1141.591,22.661,-49.918,179.885,6.321,149.181
C08570=1141.586,22.910,-49.932,179.888,6.323,149.180
C08571=1141.581,23.160,-49.947,179.890,6.324,149.180
C08572=1141.574,23.409,-49.961,179.892,6.324,149.179
C08573=1141.570,23.659,-49.975,179.895,6.326,149.179
C08574=1141.565,23.909,-49.990,179.897,6.327,149.178
C08575=1141.560,24.159,-50.004,179.900,6.327,149.177
C08576=1141.555,24.408,-50.018,179.903,6.329,149.177
C08577=1141.549,24.657,-50.032,179.905,6.329,149.176
C08578=1141.544,24.906,-50.047,179.907,6.330,149.176
C08579=1141.539,25.156,-50.061,179.910,6.332,149.175
C08580=1141.535,25.406,-50.076,179.913,6.332,149.175
C08581=1141.530,25.656,-50.090,179.915,6.333,149.174
C08582=1141.525,25.905,-50.104,179.918,6.334,149.174
C08583=1141.519,26.154,-50.118,179.920,6.335,149.173
C08584=1141.514,26.404,-50.132,179.923,6.337,149.173
C08585=1141.509,26.653,-50.147,179.926,6.337,149.172
C08586=1141.504,26.903,-50.162,179.928,6.338,149.172
C08587=1141.498,27.173,-50.177,179.931,6.339,149.171
C08588=1141.493,27.441,-50.193,179.933,6.340,149.170
C08589=1141.488,27.710,-50.209,179.937,6.341,149.170
C08590=1141.482,27.979,-50.223,179.940,6.343,149.169
C08591=1141.477,28.228,-50.239,179.942,6.343,149.169
C08592=1141.472,28.478,-50.253,179.944,6.344,149.168
C08593=1141.467,28.728,-50.267,179.947,6.346,149.168
C08594=1141.462,28.977,-50.282,179.950,6.346,149.167
C08595=1141.457,29.226,-50.297,179.952,6.347,149.167
C08596=1141.452,29.476,-50.311,179.955,6.348,149.166
C08597=1141.446,29.726,-50.326,179.957,6.349,149.165
C08598=1141.441,29.975,-50.340,179.960,6.351,149.165
C08599=1141.436,30.224,-50.355,179.963,6.351,149.164
C08600=1141.431,30.474,-50.369,179.965,6.352,149.164
C08601=1141.426,30.724,-50.383,179.968,6.354,149.163
C08602=1141.421,30.973,-50.399,179.970,6.354,149.163
C08603=1141.416,31.223,-50.413,179.973,6.356,149.162
C08604=1141.411,31.472,-50.427,179.976,6.356,149.162
C08605=1141.406,31.722,-50.442,179.978,6.357,149.161
C08606=1141.401,31.972,-50.457,179.981,6.359,149.161
C08607=1141.396,32.221,-50.472,179.983,6.359,149.160
C08608=1141.391,32.470,-50.487,179.986,6.361,149.160
C08609=1141.386,32.720,-50.501,179.988,6.362,149.159
C08610=1141.381,32.970,-50.516,179.991,6.362,149.158
C08611=1141.376,33.219,-50.531,179.994,6.364,149.158
C08612=1141.371,33.468,-50.546,179.996,6.364,149.157
C08613=1141.365,33.718,-50.561,179.999,6.366,149.157
C08614=1141.361,33.968,-50.575,-179.999,6.367,149.156
C08615=1141.356,34.217,-50.590,-179.996,6.368,149.156
C08616=1141.350,34.466,-50.604,-179.993,6.369,149.155
C08617=1141.345,34.716,-50.619,-179.991,6.370,149.155
C08618=1141.340,34.965,-50.634,-179.988,6.371,149.154
C08619=1141.335,35.214,-50.649,-179.986,6.372,149.154
C08620=1141.330,35.464,-50.663,-179.983,6.373,149.153
C08621=1141.325,35.713,-50.678,-179.980,6.374,149.153
C08622=1141.320,35.963,-50.693,-179.978,6.375,149.152
C08623=1141.315,36.213,-50.708,-179.975,6.376,149.151
C08624=1141.310,36.462,-50.723,-179.973,6.377,149.151
C08625=1141.304,36.712,-50.738,-179.970,6.378,149.151
C08626=1141.299,36.961,-50.752,-179.967,6.379,149.150
C08627=1141.295,37.211,-50.768,-179.965,6.380,149.149
C08628=1141.290,37.461,-50.783,-179.963,6.381,149.149
C08629=1141.285,37.710,-50.798,-179.959,6.382,149.148
C08630=1141.280,37.960,-50.813,-179.957,6.383,149.148
C08631=1141.275,38.209,-50.828,-179.954,6.384,149.147
C08632=1141.270,38.459,-50.843,-179.952,6.385,149.147
C08633=1141.264,38.709,-50.857,-179.950,6.386,149.146
C08634=1141.260,38.958,-50.872,-179.946,6.387,149.146
C08635=1141.254,39.207,-50.888,-179.944,6.388,149.145
C08636=1141.249,39.457,-50.902,-179.941,6.390,149.145
C08637=1141.244,39.706,-50.918,-179.939,6.390,149.144
C08638=1141.239,39.955,-50.933,-179.936,6.392,149.144
C08639=1141.234,40.205,-50.948,-179.934,6.393,149.143
C08640=1141.229,40.454,-50.963,-179.931,6.394,149.142
C08641=1141.224,40.704,-50.978,-179.928,6.395,149.142
C08642=1141.219,40.953,-50.993,-179.925,6.396,149.141
C08643=1141.215,41.203,-51.008,-179.923,6.397,149.141
C08644=1141.209,41.453,-51.024,-179.921,6.398,149.140
C08645=1141.205,41.702,-51.039,-179.918,6.399,149.140
C08646=1141.199,41.952,-51.053,-179.915,6.400,149.139
C08647=1141.193,42.201,-51.069,-179.913,6.402,149.139
C08648=1141.189,42.450,-51.084,-179.910,6.402,149.138
C08649=1141.183,42.700,-51.100,-179.907,6.404,149.138
C08650=1141.178,42.949,-51.114,-179.905,6.405,149.137
C08651=1141.173,43.199,-51.129,-179.902,6.406,149.137
C08652=1141.169,43.449,-51.145,-179.900,6.407,149.136
C08653=1141.164,43.698,-51.160,-179.897,6.408,149.136
C08654=1141.159,43.947,-51.175,-179.894,6.409,149.135
C08655=1141.153,44.197,-51.190,-179.892,6.410,149.135
C08656=1141.149,44.446,-51.205,-179.889,6.411,149.134
C08657=1141.143,44.696,-51.221,-179.886,6.412,149.133
C08658=1141.138,44.946,-51.237,-179.884,6.413,149.133
C08659=1141.134,45.195,-51.252,-179.881,6.415,149.132
C08660=1141.128,45.444,-51.267,-179.879,6.415,149.132
C08661=1141.124,45.693,-51.282,-179.876,6.417,149.131
C08662=1141.118,45.943,-51.297,-179.873,6.417,149.131
C08663=1141.113,46.193,-51.313,-179.870,6.419,149.130
C08664=1141.109,46.442,-51.328,-179.868,6.420,149.130
C08665=1141.103,46.692,-51.344,-179.865,6.421,149.129
C08666=1141.098,46.941,-51.359,-179.863,6.422,149.129
C08667=1141.093,47.190,-51.374,-179.860,6.424,149.128
C08668=1141.088,47.440,-51.390,-179.857,6.424,149.128
C08669=1141.084,47.690,-51.405,-179.855,6.426,149.127
C08670=1141.078,47.939,-51.421,-179.853,6.427,149.127
C08671=1141.073,48.188,-51.436,-179.849,6.428,149.126
C08672=1141.068,48.438,-51.452,-179.847,6.429,149.126
C08673=1141.064,48.688,-51.467,-179.844,6.430,149.125
C08674=1141.058,48.937,-51.483,-179.842,6.431,149.125
C08675=1141.053,49.186,-51.499,-179.839,6.432,149.124
C08676=1141.048,49.435,-51.514,-179.837,6.433,149.124
C08677=1141.043,49.686,-51.530,-179.834,6.435,149.123
C08678=1141.038,49.935,-51.545,-179.831,6.436,149.123
C08679=1141.033,50.184,-51.560,-179.829,6.437,149.122
C08680=1141.028,50.433,-51.576,-179.825,6.438,149.121
C08681=1141.023,50.684,-51.592,-179.823,6.439,149.121
C08682=1141.018,50.933,-51.607,-179.821,6.441,149.121
C08683=1141.013,51.182,-51.622,-179.818,6.441,149.120
C08684=1141.008,51.431,-51.639,-179.815,6.443,149.119
C08685=1141.003,51.681,-51.654,-179.813,6.444,149.119
C08686=1140.998,51.930,-51.670,-179.810,6.445,149.118
C08687=1140.993,52.179,-51.685,-179.808,6.446,149.118
C08688=1140.988,52.430,-51.701,-179.805,6.448,149.117
C08689=1140.983,52.679,-51.717,-179.802,6.448,149.117
C08690=1140.978,52.928,-51.732,-179.799,6.450,149.116
C08691=1140.972,53.197,-51.749,-179.796,6.451,149.116
C08692=1140.967,53.466,-51.767,-179.793,6.453,149.115
C08693=1140.962,53.735,-51.784,-179.791,6.453,149.115
C08694=1140.957,54.003,-51.800,-179.788,6.455,149.114
C08695=1140.951,54.252,-51.816,-179.785,6.456,149.114
C08696=1140.947,54.502,-51.832,-179.783,6.457,149.113
C08697=1140.942,54.751,-51.848,-179.780,6.458,149.113
C08698=1140.936,55.000,-51.863,-179.778,6.459,149.112
C08699=1140.931,55.250,-51.879,-179.775,6.461,149.111
C08700=1140.926,55.500,-51.895,-179.772,6.461,149.111
C08701=1140.922,55.748,-51.911,-179.770,6.463,149.111
C08702=1140.917,55.998,-51.927,-179.766,6.464,149.110
C08703=1140.911,56.248,-51.942,-179.764,6.465,149.109
C08704=1140.906,56.497,-51.959,-179.761,6.467,149.109
C08705=1140.902,56.747,-51.975,-179.759,6.467,149.108
C08706=1140.896,56.996,-51.990,-179.756,6.469,149.108
C08707=1140.891,57.246,-52.006,-179.753,6.471,149.108
C08708=1140.886,57.495,-52.022,-179.751,6.471,149.107
C08709=1140.881,57.744,-52.038,-179.748,6.473,149.106
C08710=1140.876,57.994,-52.055,-179.746,6.473,149.106
C08711=1140.871,58.243,-52.070,-179.743,6.475,149.106
C08712=1140.866,58.493,-52.086,-179.740,6.476,149.105
C08713=1140.861,58.742,-52.102,-179.738,6.477,149.104
C08714=1140.856,58.992,-52.118,-179.735,6.479,149.104
C08715=1140.851,59.242,-52.134,-179.732,6.479,149.103
C08716=1140.846,59.490,-52.150,-179.729,6.481,149.103
C08717=1140.841,59.741,-52.166,-179.727,6.482,149.102
C08718=1140.836,59.989,-52.183,-179.724,6.483,149.102
C08719=1140.831,60.239,-52.198,-179.721,6.485,149.101
C08720=1140.826,60.488,-52.215,-179.719,6.486,149.101
C08721=1140.821,60.738,-52.230,-179.716,6.487,149.100
C08722=1140.816,60.987,-52.247,-179.714,6.488,149.100
C08723=1140.811,61.237,-52.263,-179.711,6.489,149.099
C08724=1140.806,61.486,-52.279,-179.708,6.491,149.099
C08725=1140.801,61.735,-52.295,-179.706,6.492,149.098
C08726=1140.797,61.985,-52.312,-179.703,6.493,149.098
C08727=1140.791,62.234,-52.327,-179.700,6.495,149.097
C08728=1140.787,62.484,-52.344,-179.698,6.495,149.097
C08729=1140.781,62.733,-52.359,-179.695,6.497,149.096
C08730=1140.777,62.983,-52.376,-179.693,6.498,149.096
C08731=1140.771,63.232,-52.392,-179.689,6.499,149.095
C08732=1140.767,63.482,-52.408,-179.687,6.501,149.095
C08733=1140.762,63.730,-52.425,-179.684,6.502,149.094
C08734=1140.757,63.980,-52.441,-179.682,6.503,149.094
C08735=1140.752,64.229,-52.457,-179.678,6.504,149.093
C08736=1140.747,64.480,-52.473,-179.676,6.505,149.093
C08737=1140.741,64.728,-52.490,-179.674,6.507,149.092
C08738=1140.737,64.978,-52.506,-179.671,6.507,149.092
C08739=1140.732,65.227,-52.522,-179.668,6.509,149.091
C08740=1140.727,65.477,-52.539,-179.665,6.511,149.091
C08741=1140.722,65.726,-52.555,-179.663,6.511,149.090
C08742=1140.717,65.976,-52.571,-179.660,6.513,149.090
C08743=1140.711,66.225,-52.588,-179.657,6.515,149.089
C08744=1140.707,66.474,-52.605,-179.655,6.515,149.089
C08745=1140.702,66.724,-52.620,-179.652,6.517,149.088
C08746=1140.697,66.973,-52.637,-179.649,6.518,149.088
C08747=1140.693,67.223,-52.653,-179.647,6.519,149.087
C08748=1140.688,67.471,-52.670,-179.644,6.520,149.087
C08749=1140.682,67.722,-52.686,-179.641,6.522,149.086
C08750=1140.677,67.971,-52.703,-179.639,6.523,149.086
C08751=1140.672,68.220,-52.719,-179.636,6.525,149.085
C08752=1140.668,68.470,-52.736,-179.633,6.526,149.085
C08753=1140.662,68.719,-52.753,-179.631,6.527,149.084
C08754=1140.657,68.969,-52.769,-179.628,6.528,149.084
C08755=1140.652,69.218,-52.785,-179.625,6.530,149.083
C08756=1140.648,69.467,-52.802,-179.623,6.531,149.083
C08757=1140.643,69.717,-52.819,-179.620,6.532,149.082
C08758=1140.637,69.966,-52.835,-179.617,6.534,149.082
C08759=1140.633,70.216,-52.851,-179.615,6.534,149.081
C08760=1140.628,70.465,-52.868,-179.612,6.536,149.081
C08761=1140.622,70.714,-52.885,-179.609,6.538,149.080
C08762=1140.618,70.964,-52.902,-179.607,6.538,149.080
C08763=1140.613,71.213,-52.918,-179.604,6.540,149.079
C08764=1140.608,71.462,-52.935,-179.601,6.541,149.079
C08765=1140.603,71.712,-52.952,-179.599,6.542,149.078
C08766=1140.598,71.961,-52.968,-179.596,6.544,149.078
C08767=1140.593,72.210,-52.985,-179.593,6.545,149.077
C08768=1140.588,72.460,-53.002,-179.590,6.547,149.077
C08769=1140.583,72.709,-53.018,-179.588,6.548,149.076
C08770=1140.578,72.959,-53.035,-179.585,6.549,149.076
C08771=1140.573,73.209,-53.052,-179.582,6.551,149.075
C08772=1140.568,73.457,-53.068,-179.580,6.552,149.075
C08773=1140.563,73.707,-53.085,-179.577,6.553,149.074
C08774=1140.558,73.957,-53.102,-179.574,6.554,149.074
C08775=1140.553,74.206,-53.119,-179.572,6.555,149.073
C08776=1140.548,74.455,-53.135,-179.569,6.557,149.073
C08777=1140.544,74.704,-53.153,-179.566,6.559,149.073
C08778=1140.539,74.954,-53.170,-179.563,6.560,149.072
C08779=1140.534,75.203,-53.186,-179.561,6.561,149.071
C08780=1140.529,75.452,-53.204,-179.558,6.562,149.071
C08781=1140.524,75.702,-53.220,-179.555,6.564,149.071
C08782=1140.519,75.952,-53.237,-179.553,6.565,149.070
C08783=1140.514,76.201,-53.254,-179.550,6.566,149.069
C08784=1140.509,76.450,-53.270,-179.547,6.568,149.069
C08785=1140.504,76.700,-53.288,-179.544,6.570,149.069
C08786=1140.500,76.949,-53.304,-179.542,6.570,149.068
C08787=1140.494,77.198,-53.321,-179.539,6.572,149.068
C08788=1140.490,77.447,-53.339,-179.536,6.573,149.067
C08789=1140.484,77.697,-53.356,-179.534,6.575,149.067
C08790=1140.480,77.947,-53.373,-179.531,6.576,149.066
C08791=1140.474,78.196,-53.390,-179.528,6.577,149.066
C08792=1140.470,78.445,-53.406,-179.525,6.579,149.065
C08793=1140.464,78.695,-53.423,-179.523,6.580,149.065
C08794=1140.460,78.944,-53.441,-179.520,6.581,149.064
C08795=1140.454,79.212,-53.459,-179.517,6.583,149.064
C08796=1140.449,79.481,-53.478,-179.514,6.584,149.063
C08797=1140.444,79.749,-53.496,-179.511,6.586,149.063
C08798=1140.438,80.018,-53.514,-179.509,6.587,149.062
C08799=1140.434,80.267,-53.531,-179.505,6.589,149.061
C08800=1140.429,80.516,-53.549,-179.503,6.590,149.061
C08801=1140.424,80.766,-53.566,-179.500,6.591,149.061
C08802=1140.418,81.015,-53.582,-179.498,6.593,149.060
C08803=1140.413,81.265,-53.600,-179.494,6.594,149.060
C08804=1140.409,81.513,-53.617,-179.492,6.596,149.059
C08805=1140.404,81.763,-53.634,-179.490,6.597,149.059
C08806=1140.399,82.013,-53.652,-179.487,6.598,149.058
C08807=1140.394,82.262,-53.669,-179.484,6.600,149.058
C08808=1140.389,82.511,-53.686,-179.481,6.601,149.057
C08809=1140.384,82.760,-53.704,-179.479,6.602,149.057
C08810=1140.379,83.010,-53.721,-179.476,6.604,149.056
C08811=1140.374,83.259,-53.738,-179.473,6.605,149.056
C08812=1140.370,83.508,-53.755,-179.470,6.607,149.055
C08813=1140.365,83.758,-53.773,-179.467,6.608,149.055
C08814=1140.360,84.007,-53.790,-179.465,6.609,149.054
C08815=1140.355,84.257,-53.808,-179.462,6.611,149.054
C08816=1140.349,84.506,-53.824,-179.460,6.613,149.054
C08817=1140.345,84.755,-53.842,-179.456,6.614,149.053
C08818=1140.339,85.005,-53.859,-179.454,6.615,149.052
C08819=1140.335,85.254,-53.877,-179.452,6.616,149.052
C08820=1140.330,85.504,-53.894,-179.449,6.618,149.052
C08821=1140.325,85.753,-53.912,-179.446,6.619,149.051
C08822=1140.321,86.002,-53.929,-179.443,6.621,149.051
C08823=1140.316,86.251,-53.947,-179.441,6.622,149.050
C08824=1140.310,86.501,-53.964,-179.438,6.623,149.050
C08825=1140.305,86.750,-53.982,-179.435,6.625,149.049
C08826=1140.301,87.000,-53.998,-179.432,6.626,149.049
C08827=1140.296,87.249,-54.016,-179.429,6.628,149.048
C08828=1140.290,87.498,-54.033,-179.427,6.629,149.048
C08829=1140.285,87.747,-54.051,-179.424,6.631,149.047
C08830=1140.280,87.996,-54.069,-179.422,6.632,149.047
C08831=1140.276,88.246,-54.086,-179.418,6.634,149.046
C08832=1140.271,88.495,-54.104,-179.416,6.635,149.046
C08833=1140.266,88.745,-54.121,-179.414,6.636,149.045
C08834=1140.261,88.994,-54.139,-179.411,6.638,149.045
C08835=1140.256,89.243,-54.157,-179.408,6.639,149.045
C08836=1140.252,89.493,-54.174,-179.405,6.641,149.044
C08837=1140.247,89.742,-54.192,-179.402,6.642,149.044
C08838=1140.242,89.991,-54.210,-179.399,6.644,149.043
C08839=1140.236,90.241,-54.227,-179.397,6.645,149.043
C08840=1140.232,90.490,-54.245,-179.394,6.647,149.042
C08841=1140.227,90.739,-54.263,-179.391,6.648,149.042
C08842=1140.222,90.988,-54.281,-179.389,6.650,149.041
C08843=1140.217,91.238,-54.298,-179.386,6.651,149.041
C08844=1140.212,91.487,-54.316,-179.383,6.653,149.040
C08845=1140.207,91.736,-54.334,-179.381,6.654,149.040
C08846=1140.202,91.986,-54.351,-179.378,6.655,149.039
C08847=1140.197,92.235,-54.369,-179.375,6.657,149.039
C08848=1140.192,92.484,-54.387,-179.372,6.658,149.038
C08849=1140.187,92.734,-54.405,-179.369,6.660,149.038
C08850=1140.183,92.983,-54.423,-179.367,6.662,149.038
C08851=1140.178,93.233,-54.440,-179.365,6.663,149.037
C08852=1140.173,93.482,-54.458,-179.361,6.664,149.037
C08853=1140.168,93.732,-54.476,-179.359,6.666,149.036
C08854=1140.163,93.981,-54.494,-179.356,6.667,149.036
C08855=1140.158,94.230,-54.512,-179.353,6.669,149.035
C08856=1140.153,94.479,-54.530,-179.350,6.671,149.035
C08857=1140.148,94.729,-54.548,-179.347,6.672,149.034
C08858=1140.143,94.978,-54.566,-179.345,6.673,149.034
C08859=1140.138,95.227,-54.584,-179.342,6.675,149.033
C08860=1140.133,95.476,-54.602,-179.340,6.676,149.033
C08861=1140.129,95.726,-54.620,-179.337,6.678,149.033
C08862=1140.124,95.975,-54.638,-179.334,6.680,149.032
C08863=1140.119,96.225,-54.656,-179.331,6.681,149.032
C08864=1140.114,96.474,-54.674,-179.328,6.683,149.031
C08865=1140.109,96.723,-54.692,-179.325,6.684,149.031
C08866=1140.105,96.972,-54.710,-179.323,6.685,149.030
C08867=1140.100,97.221,-54.728,-179.321,6.687,149.030
C08868=1140.095,97.471,-54.746,-179.318,6.688,149.029
C08869=1140.090,97.720,-54.764,-179.315,6.690,149.029
C08870=1140.086,97.970,-54.782,-179.312,6.691,149.028
C08871=1140.081,98.219,-54.800,-179.309,6.693,149.028
C08872=1140.076,98.468,-54.818,-179.306,6.695,149.028
C08873=1140.071,98.717,-54.836,-179.304,6.696,149.027
C08874=1140.066,98.966,-54.854,-179.301,6.698,149.027
C08875=1140.060,99.216,-54.873,-179.299,6.699,149.026
C08876=1140.056,99.466,-54.891,-179.296,6.700,149.026
C08877=1140.051,99.715,-54.909,-179.293,6.702,149.025
C08878=1140.046,99.964,-54.927,-179.290,6.704,149.025
C08879=1140.041,100.213,-54.945,-179.287,6.705,149.024
C08880=1140.037,100.462,-54.964,-179.285,6.707,149.024
C08881=1140.032,100.711,-54.982,-179.282,6.709,149.024
C08882=1140.027,100.961,-55.001,-179.279,6.710,149.023
C08883=1140.022,101.210,-55.018,-179.276,6.712,149.023
C08884=1140.017,101.459,-55.036,-179.273,6.713,149.022
C08885=1140.012,101.709,-55.054,-179.270,6.715,149.022
C08886=1140.008,101.958,-55.073,-179.268,6.716,149.021
C08887=1140.002,102.207,-55.092,-179.266,6.718,149.021
C08888=1139.997,102.457,-55.110,-179.263,6.719,149.020
C08889=1139.992,102.706,-55.128,-179.260,6.721,149.020
C08890=1139.987,102.955,-55.146,-179.257,6.722,149.019
C08891=1139.983,103.204,-55.165,-179.254,6.724,149.019
C08892=1139.978,103.454,-55.184,-179.251,6.726,149.019
C08893=1139.973,103.703,-55.202,-179.249,6.727,149.018
C08894=1139.969,103.953,-55.220,-179.246,6.729,149.018
C08895=1139.964,104.201,-55.239,-179.243,6.731,149.017
C08896=1139.958,104.451,-55.257,-179.240,6.732,149.017
C08897=1139.953,104.700,-55.275,-179.238,6.734,149.016
C08898=1139.949,104.950,-55.294,-179.235,6.735,149.016
C08899=1139.944,105.218,-55.314,-179.232,6.737,149.015
C08900=1139.939,105.486,-55.334,-179.229,6.739,149.015
C08901=1139.933,105.755,-55.354,-179.226,6.740,149.015
C08902=1139.928,106.023,-55.373,-179.223,6.742,149.014
C08903=1139.924,106.272,-55.392,-179.220,6.743,149.014
C08904=1139.918,106.522,-55.411,-179.218,6.745,149.013
C08905=1139.913,106.770,-55.429,-179.215,6.747,149.013
C08906=1139.908,107.020,-55.448,-179.212,6.748,149.012
C08907=1139.903,107.269,-55.466,-179.209,6.750,149.012
C08908=1139.899,107.518,-55.485,-179.207,6.752,149.012
C08909=1139.894,107.768,-55.504,-179.204,6.753,149.011
C08910=1139.889,108.017,-55.523,-179.201,6.755,149.010
C08911=1139.884,108.266,-55.541,-179.198,6.756,149.010
C08912=1139.879,108.515,-55.560,-179.195,6.758,149.010
C08913=1139.875,108.765,-55.578,-179.193,6.760,149.009
C08914=1139.869,109.014,-55.598,-179.190,6.761,149.009
C08915=1139.865,109.263,-55.616,-179.187,6.763,149.008
C08916=1139.860,109.512,-55.635,-179.184,6.765,149.008
C08917=1139.855,109.762,-55.654,-179.182,6.766,149.008
C08918=1139.851,110.011,-55.672,-179.179,6.768,149.007
C08919=1139.845,110.260,-55.691,-179.176,6.770,149.007
C08920=1139.841,110.509,-55.710,-179.173,6.771,149.006
C08921=1139.835,110.759,-55.729,-179.170,6.773,149.006
C08922=1139.831,111.008,-55.748,-179.168,6.774,149.005
C08923=1139.826,111.257,-55.767,-179.165,6.776,149.005
C08924=1139.821,111.506,-55.785,-179.162,6.778,149.005
C08925=1139.816,111.756,-55.804,-179.159,6.780,149.004
C08926=1139.811,112.005,-55.822,-179.157,6.781,149.004
C08927=1139.807,112.255,-55.842,-179.154,6.783,149.003
C08928=1139.802,112.503,-55.861,-179.151,6.785,149.003
C08929=1139.796,112.753,-55.879,-179.148,6.786,149.002
C08930=1139.792,113.002,-55.898,-179.146,6.788,149.002
C08931=1139.787,113.251,-55.918,-179.143,6.790,149.002
C08932=1139.783,113.501,-55.936,-179.140,6.791,149.001
C08933=1139.777,113.749,-55.955,-179.137,6.793,149.001
C08934=1139.773,113.999,-55.974,-179.134,6.794,149.000
C08935=1139.768,114.248,-55.993,-179.132,6.796,149.000
C08936=1139.763,114.498,-56.013,-179.129,6.798,148.999
C08937=1139.758,114.746,-56.031,-179.126,6.799,148.999
C08938=1139.754,114.996,-56.051,-179.123,6.801,148.999
C08939=1139.749,115.245,-56.069,-179.121,6.803,148.998
C08940=1139.743,115.494,-56.088,-179.118,6.804,148.998
C08941=1139.739,115.744,-56.108,-179.115,6.806,148.997
C08942=1139.734,115.992,-56.127,-179.112,6.808,148.997
C08943=1139.729,116.242,-56.146,-179.110,6.810,148.997
C08944=1139.724,116.491,-56.164,-179.107,6.811,148.996
C08945=1139.720,116.740,-56.184,-179.104,6.813,148.996
C08946=1139.715,116.990,-56.204,-179.102,6.815,148.995
C08947=1139.710,117.239,-56.222,-179.098,6.816,148.995
C08948=1139.706,117.488,-56.242,-179.096,6.818,148.994
C08949=1139.700,117.737,-56.261,-179.093,6.819,148.994
C08950=1139.696,117.986,-56.280,-179.090,6.821,148.994
C08951=1139.691,118.235,-56.300,-179.087,6.823,148.993
C08952=1139.686,118.485,-56.319,-179.085,6.824,148.993
C08953=1139.681,118.734,-56.338,-179.082,6.826,148.992
C08954=1139.677,118.983,-56.357,-179.079,6.828,148.992
C08955=1139.671,119.232,-56.376,-179.077,6.829,148.991
C08956=1139.666,119.482,-56.396,-179.074,6.831,148.991
C08957=1139.662,119.731,-56.415,-179.071,6.833,148.991
C08958=1139.657,119.980,-56.434,-179.068,6.834,148.990
C08959=1139.652,120.230,-56.454,-179.066,6.836,148.990
C08960=1139.647,120.478,-56.473,-179.062,6.839,148.989
C08961=1139.643,120.728,-56.492,-179.060,6.840,148.989
C08962=1139.638,120.977,-56.511,-179.057,6.842,148.989
C08963=1139.633,121.226,-56.531,-179.054,6.844,148.988
C08964=1139.628,121.476,-56.551,-179.051,6.845,148.988
C08965=1139.623,121.725,-56.570,-179.049,6.847,148.987
C08966=1139.619,121.974,-56.589,-179.046,6.849,148.987
C08967=1139.614,122.223,-56.610,-179.043,6.850,148.987
C08968=1139.609,122.472,-56.629,-179.041,6.852,148.986
C08969=1139.604,122.721,-56.648,-179.038,6.854,148.986
C08970=1139.599,122.970,-56.668,-179.035,6.856,148.985
C08971=1139.595,123.219,-56.687,-179.032,6.857,148.985
C08972=1139.590,123.469,-56.706,-179.030,6.859,148.985
C08973=1139.585,123.718,-56.726,-179.027,6.861,148.984
C08974=1139.580,123.967,-56.745,-179.024,6.863,148.984
C08975=1139.576,124.216,-56.766,-179.021,6.865,148.983
C08976=1139.570,124.465,-56.785,-179.018,6.867,148.983
C08977=1139.566,124.715,-56.805,-179.015,6.868,148.983
C08978=1139.561,124.964,-56.824,-179.013,6.870,148.982
C08979=1139.556,125.213,-56.843,-179.010,6.872,148.982
C08980=1139.552,125.462,-56.863,-179.007,6.873,148.981
C08981=1139.547,125.711,-56.883,-179.005,6.875,148.981
C08982=1139.542,125.961,-56.903,-179.002,6.877,148.981
C08983=1139.537,126.210,-56.922,-178.999,6.878,148.980
C08984=1139.533,126.459,-56.942,-178.996,6.881,148.980
C08985=1139.528,126.708,-56.962,-178.993,6.883,148.979
C08986=1139.522,126.957,-56.981,-178.990,6.884,148.979
C08987=1139.518,127.206,-57.002,-178.988,6.886,148.979
C08988=1139.513,127.456,-57.021,-178.985,6.888,148.978
C08989=1139.509,127.705,-57.041,-178.982,6.889,148.978
C08990=1139.503,127.953,-57.061,-178.979,6.891,148.977
C08991=1139.499,128.203,-57.081,-178.977,6.893,148.977
C08992=1139.494,128.453,-57.100,-178.974,6.894,148.977
C08993=1139.490,128.702,-57.121,-178.971,6.897,148.976
C08994=1139.484,128.950,-57.140,-178.968,6.899,148.976
C08995=1139.479,129.200,-57.160,-178.965,6.900,148.976
C08996=1139.475,129.449,-57.180,-178.962,6.902,148.975
C08997=1139.470,129.699,-57.200,-178.960,6.904,148.975
C08998=1139.465,129.947,-57.220,-178.957,6.905,148.974
C08999=1139.460,130.196,-57.239,-178.954,6.907,148.974
C09000=1139.456,130.445,-57.260,-178.952,6.909,148.974
C09001=1139.451,130.695,-57.279,-178.948,6.911,148.973
C09002=1139.447,130.944,-57.299,-178.946,6.913,148.973
C09003=1139.441,131.213,-57.321,-178.943,6.915,148.972
C09004=1139.436,131.481,-57.342,-178.940,6.917,148.972
C09005=1139.430,131.750,-57.364,-178.937,6.919,148.972
C09006=1139.425,132.018,-57.386,-178.934,6.920,148.971
C09007=1139.421,132.267,-57.405,-178.931,6.922,148.971
C09008=1139.416,132.516,-57.426,-178.928,6.924,148.970
C09009=1139.412,132.766,-57.445,-178.925,6.926,148.970
C09010=1139.406,133.015,-57.466,-178.923,6.928,148.970
C09011=1139.402,133.264,-57.487,-178.920,6.930,148.969
C09012=1139.397,133.513,-57.506,-178.917,6.932,148.969
C09013=1139.392,133.762,-57.526,-178.914,6.933,148.968
C09014=1139.387,134.011,-57.546,-178.911,6.936,148.968
C09015=1139.383,134.260,-57.566,-178.908,6.937,148.968
C09016=1139.378,134.510,-57.587,-178.906,6.939,148.967
C09017=1139.373,134.759,-57.607,-178.903,6.941,148.967
C09018=1139.369,135.008,-57.627,-178.900,6.943,148.966
C09019=1139.364,135.257,-57.648,-178.898,6.944,148.966
C09020=1139.358,135.506,-57.668,-178.894,6.947,148.966
C09021=1139.354,135.755,-57.688,-178.892,6.948,148.965
C09022=1139.349,136.004,-57.708,-178.889,6.950,148.965
C09023=1139.344,136.254,-57.728,-178.886,6.952,148.965
C09024=1139.339,136.503,-57.749,-178.883,6.954,148.964
C09025=1139.335,136.752,-57.769,-178.880,6.956,148.964
C09026=1139.330,137.001,-57.790,-178.878,6.958,148.964
C09027=1139.326,137.250,-57.809,-178.875,6.960,148.963
C09028=1139.320,137.500,-57.830,-178.872,6.962,148.963
C09029=1139.316,137.749,-57.851,-178.870,6.963,148.962
C09030=1139.312,137.998,-57.871,-178.866,6.966,148.962
C09031=1139.306,138.247,-57.892,-178.864,6.967,148.962
C09032=1139.301,138.495,-57.912,-178.861,6.969,148.961
C09033=1139.297,138.745,-57.932,-178.858,6.971,148.961
C09034=1139.292,138.994,-57.952,-178.855,6.973,148.960
C09035=1139.287,139.243,-57.973,-178.852,6.975,148.960
C09036=1139.283,139.492,-57.993,-178.849,6.977,148.960
C09037=1139.277,139.741,-58.014,-178.847,6.978,148.959
C09038=1139.273,139.990,-58.035,-178.844,6.981,148.959
C09039=1139.269,140.239,-58.055,-178.842,6.982,148.959
C09040=1139.263,140.488,-58.076,-178.838,6.985,148.958
C09041=1139.259,140.738,-58.096,-178.836,6.986,148.958
C09042=1139.254,140.987,-58.116,-178.833,6.988,148.958
C09043=1139.249,141.236,-58.137,-178.830,6.990,148.957
C09044=1139.245,141.485,-58.158,-178.828,6.992,148.957
C09045=1139.239,141.734,-58.178,-178.824,6.994,148.956
C09046=1139.235,141.983,-58.199,-178.822,6.996,148.956
C09047=1139.231,142.232,-58.219,-178.819,6.997,148.956
C09048=1139.225,142.481,-58.240,-178.817,7.000,148.955
C09049=1139.221,142.730,-58.261,-178.813,7.002,148.955
C09050=1139.216,142.980,-58.282,-178.811,7.004,148.955
C09051=1139.212,143.229,-58.302,-178.808,7.005,148.954
C09052=1139.207,143.478,-58.324,-178.805,7.007,148.954
C09053=1139.203,143.727,-58.344,-178.802,7.010,148.954
C09054=1139.197,143.976,-58.365,-178.799,7.011,148.953
C09055=1139.193,144.225,-58.386,-178.796,7.013,148.953
C09056=1139.188,144.474,-58.407,-178.794,7.015,148.952
C09057=1139.183,144.723,-58.427,-178.791,7.018,148.952
C09058=1139.178,144.972,-58.448,-178.788,7.019,148.952
C09059=1139.174,145.221,-58.468,-178.785,7.021,148.951
C09060=1139.169,145.471,-58.489,-178.783,7.023,148.951
C09061=1139.164,145.719,-58.510,-178.779,7.025,148.951
C09062=1139.159,145.968,-58.531,-178.777,7.027,148.950
C09063=1139.155,146.218,-58.552,-178.774,7.029,148.950
C09064=1139.150,146.467,-58.573,-178.772,7.031,148.950
C09065=1139.145,146.716,-58.594,-178.768,7.033,148.949
C09066=1139.141,146.965,-58.615,-178.766,7.035,148.949
C09067=1139.136,147.214,-58.636,-178.763,7.037,148.949
C09068=1139.131,147.463,-58.656,-178.760,7.038,148.948
C09069=1139.126,147.712,-58.677,-178.757,7.041,148.948
C09070=1139.121,147.961,-58.699,-178.754,7.043,148.947
C09071=1139.117,148.211,-58.720,-178.752,7.045,148.947
C09072=1139.112,148.460,-58.741,-178.749,7.047,148.947
C09073=1139.108,148.709,-58.761,-178.746,7.049,148.947
C09074=1139.103,148.957,-58.783,-178.743,7.051,148.946
C09075=1139.098,149.207,-58.804,-178.741,7.052,148.946
C09076=1139.093,149.456,-58.824,-178.737,7.055,148.945
C09077=1139.089,149.705,-58.846,-178.735,7.057,148.945
C09078=1139.084,149.954,-58.867,-178.732,7.059,148.945
C09079=1139.079,150.203,-58.889,-178.729,7.061,148.945
C09080=1139.075,150.452,-58.909,-178.726,7.063,148.944
C09081=1139.069,150.701,-58.930,-178.724,7.065,148.944
C09082=1139.065,150.950,-58.952,-178.720,7.067,148.943
C09083=1139.061,151.199,-58.973,-178.718,7.069,148.943
C09084=1139.056,151.448,-58.994,-178.715,7.071,148.943
C09085=1139.051,151.697,-59.015,-178.713,7.073,148.942
C09086=1139.046,151.946,-59.037,-178.709,7.075,148.942
C09087=1139.042,152.196,-59.058,-178.707,7.077,148.942
C09088=1139.037,152.445,-59.079,-178.704,7.078,148.941
C09089=1139.032,152.693,-59.100,-178.701,7.081,148.941
C09090=1139.027,152.943,-59.121,-178.698,7.083,148.941
C09091=1139.023,153.192,-59.143,-178.696,7.085,148.940
C09092=1139.018,153.440,-59.164,-178.692,7.087,148.940
C09093=1139.013,153.690,-59.185,-178.690,7.089,148.940
C09094=1139.008,153.938,-59.207,-178.687,7.091,148.939
C09095=1139.004,154.188,-59.228,-178.684,7.094,148.939
C09096=1138.999,154.437,-59.250,-178.681,7.095,148.939
C09097=1138.994,154.686,-59.271,-178.679,7.097,148.938
C09098=1138.990,154.934,-59.292,-178.675,7.100,148.938
C09099=1138.985,155.184,-59.314,-178.673,7.102,148.938
C09100=1138.980,155.433,-59.335,-178.670,7.103,148.937
C09101=1138.975,155.682,-59.357,-178.667,7.106,148.937
C09102=1138.971,155.931,-59.379,-178.664,7.108,148.937
C09103=1138.966,156.180,-59.400,-178.662,7.109,148.936
C09104=1138.961,156.429,-59.422,-178.659,7.112,148.936
C09105=1138.957,156.678,-59.443,-178.656,7.114,148.936
C09106=1138.952,156.927,-59.464,-178.653,7.116,148.935
C09107=1138.947,157.196,-59.488,-178.650,7.118,148.935
C09108=1138.942,157.465,-59.511,-178.647,7.121,148.935
C09109=1138.937,157.734,-59.534,-178.644,7.122,148.934
C09110=1138.932,158.003,-59.558,-178.641,7.125,148.934
C09111=1138.927,158.252,-59.579,-178.639,7.127,148.934
C09112=1138.922,158.501,-59.600,-178.635,7.129,148.933
C09113=1138.918,158.750,-59.622,-178.633,7.131,148.933
C09114=1138.913,158.999,-59.644,-178.630,7.133,148.933
C09115=1138.909,159.248,-59.666,-178.627,7.136,148.933
C09116=1138.904,159.497,-59.687,-178.624,7.137,148.932
C09117=1138.899,159.746,-59.709,-178.622,7.139,148.932
C09118=1138.895,159.995,-59.731,-178.618,7.142,148.931
C09119=1138.890,160.244,-59.752,-178.616,7.144,148.931
C09120=1138.886,160.493,-59.775,-178.613,7.145,148.931
C09121=1138.881,160.742,-59.796,-178.610,7.148,148.931
C09122=1138.876,160.991,-59.818,-178.607,7.150,148.930
C09123=1138.871,161.240,-59.839,-178.605,7.153,148.930
C09124=1138.866,161.489,-59.861,-178.602,7.154,148.930
C09125=1138.862,161.738,-59.883,-178.599,7.156,148.929
C09126=1138.856,161.987,-59.905,-178.596,7.159,148.929
C09127=1138.852,162.237,-59.927,-178.594,7.161,148.929
C09128=1138.847,162.485,-59.949,-178.590,7.163,148.928
C09129=1138.842,162.734,-59.971,-178.588,7.165,148.928
C09130=1138.838,162.983,-59.993,-178.585,7.167,148.928
